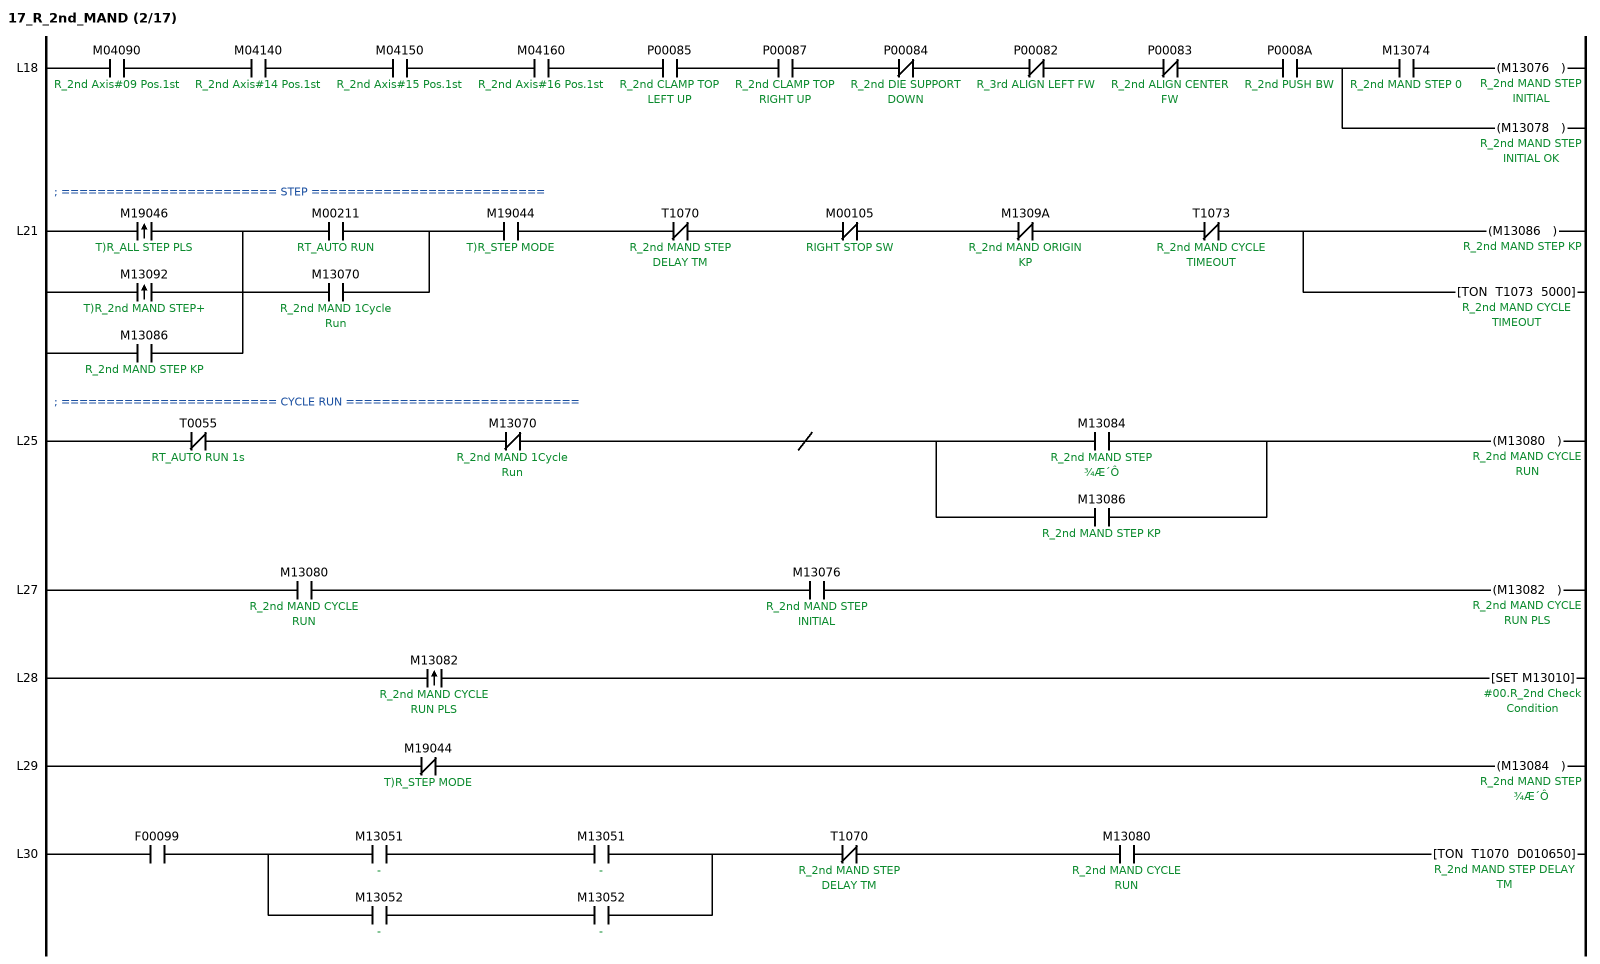
[picture p144: 17_R_2nd_MAND rungs L18-L30]
; L18
LOAD      M04090	// R_2nd Axis#09 Pos.1st
AND       M04140	// R_2nd Axis#14 Pos.1st
AND       M04150	// R_2nd Axis#15 Pos.1st
AND       M04160	// R_2nd Axis#16 Pos.1st
AND       P00085	// R_2nd CLAMP TOP LEFT UP
AND       P00087	// R_2nd CLAMP TOP RIGHT UP
AND NOT   P00084	// R_2nd DIE SUPPORT DOWN
AND NOT   P00082	// R_3rd ALIGN LEFT FW
AND NOT   P00083	// R_2nd ALIGN CENTER FW
AND       P0008A	// R_2nd PUSH BW
MPUSH
AND       M13074	// R_2nd MAND STEP 0
OUT       M13076	// R_2nd MAND STEP INITIAL
MPOP
OUT       M13078	// R_2nd MAND STEP INITIAL OK
// ======================== STEP ==========================
; L21
LOADP     M19046	// T)R_ALL STEP PLS
ORP       M13092	// T)R_2nd MAND STEP+
OR        M13086	// R_2nd MAND STEP KP
LOAD      M00211	// RT_AUTO RUN
OR        M13070	// R_2nd MAND 1Cycle Run
AND LOAD
AND       M19044	// T)R_STEP MODE
AND NOT   T1070	// R_2nd MAND STEP DELAY TM
AND NOT   M00105	// RIGHT STOP SW
AND NOT   M1309A	// R_2nd MAND ORIGIN KP
AND NOT   T1073	// R_2nd MAND CYCLE TIMEOUT
OUT       M13086	// R_2nd MAND STEP KP
TON       T1073 5000	// R_2nd MAND CYCLE TIMEOUT
// ======================== CYCLE RUN ==========================
; L25
LOAD NOT  T0055	// RT_AUTO RUN 1s
AND NOT   M13070	// R_2nd MAND 1Cycle Run
NOT
LOAD      M13084	// R_2nd MAND STEP ¾Æ´Ô
OR        M13086	// R_2nd MAND STEP KP
AND LOAD
OUT       M13080	// R_2nd MAND CYCLE RUN
; L27
LOAD      M13080	// R_2nd MAND CYCLE RUN
AND       M13076	// R_2nd MAND STEP INITIAL
OUT       M13082	// R_2nd MAND CYCLE RUN PLS
; L28
LOADP     M13082	// R_2nd MAND CYCLE RUN PLS
SET       M13010	// #00.R_2nd Check Condition
; L29
LOAD NOT  M19044	// T)R_STEP MODE
OUT       M13084	// R_2nd MAND STEP ¾Æ´Ô
; L30
LOAD      F00099
LOAD      M13051	// -
AND       M13051	// -
LOAD      M13052	// -
AND       M13052	// -
OR LOAD
AND LOAD
AND NOT   T1070	// R_2nd MAND STEP DELAY TM
AND       M13080	// R_2nd MAND CYCLE RUN
TON       T1070 D010650	// R_2nd MAND STEP DELAY TM

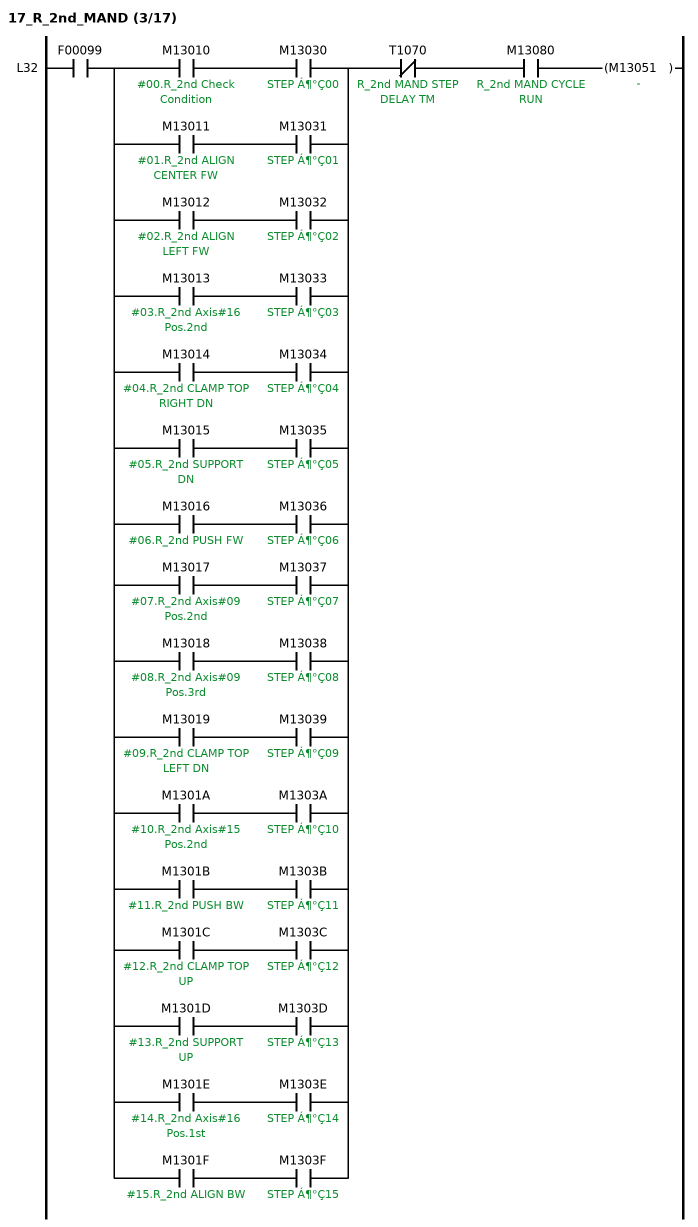
; L32
LOAD      F00099
LOAD      M13010	// #00.R_2nd Check Condition
AND       M13030	// STEP Á¶°Ç00
LOAD      M13011	// #01.R_2nd ALIGN CENTER FW
AND       M13031	// STEP Á¶°Ç01
OR LOAD
LOAD      M13012	// #02.R_2nd ALIGN LEFT FW
AND       M13032	// STEP Á¶°Ç02
OR LOAD
LOAD      M13013	// #03.R_2nd Axis#16 Pos.2nd
AND       M13033	// STEP Á¶°Ç03
OR LOAD
LOAD      M13014	// #04.R_2nd CLAMP TOP RIGHT DN
AND       M13034	// STEP Á¶°Ç04
OR LOAD
LOAD      M13015	// #05.R_2nd SUPPORT DN
AND       M13035	// STEP Á¶°Ç05
OR LOAD
LOAD      M13016	// #06.R_2nd PUSH FW
AND       M13036	// STEP Á¶°Ç06
OR LOAD
LOAD      M13017	// #07.R_2nd Axis#09 Pos.2nd
AND       M13037	// STEP Á¶°Ç07
OR LOAD
LOAD      M13018	// #08.R_2nd Axis#09 Pos.3rd
AND       M13038	// STEP Á¶°Ç08
OR LOAD
LOAD      M13019	// #09.R_2nd CLAMP TOP LEFT DN
AND       M13039	// STEP Á¶°Ç09
OR LOAD
LOAD      M1301A	// #10.R_2nd Axis#15 Pos.2nd
AND       M1303A	// STEP Á¶°Ç10
OR LOAD
LOAD      M1301B	// #11.R_2nd PUSH BW
AND       M1303B	// STEP Á¶°Ç11
OR LOAD
LOAD      M1301C	// #12.R_2nd CLAMP TOP UP
AND       M1303C	// STEP Á¶°Ç12
OR LOAD
LOAD      M1301D	// #13.R_2nd SUPPORT UP
AND       M1303D	// STEP Á¶°Ç13
OR LOAD
LOAD      M1301E	// #14.R_2nd Axis#16 Pos.1st
AND       M1303E	// STEP Á¶°Ç14
OR LOAD
LOAD      M1301F	// #15.R_2nd ALIGN BW
AND       M1303F	// STEP Á¶°Ç15
OR LOAD
AND LOAD
AND NOT   T1070	// R_2nd MAND STEP DELAY TM
AND       M13080	// R_2nd MAND CYCLE RUN
OUT       M13051	// -

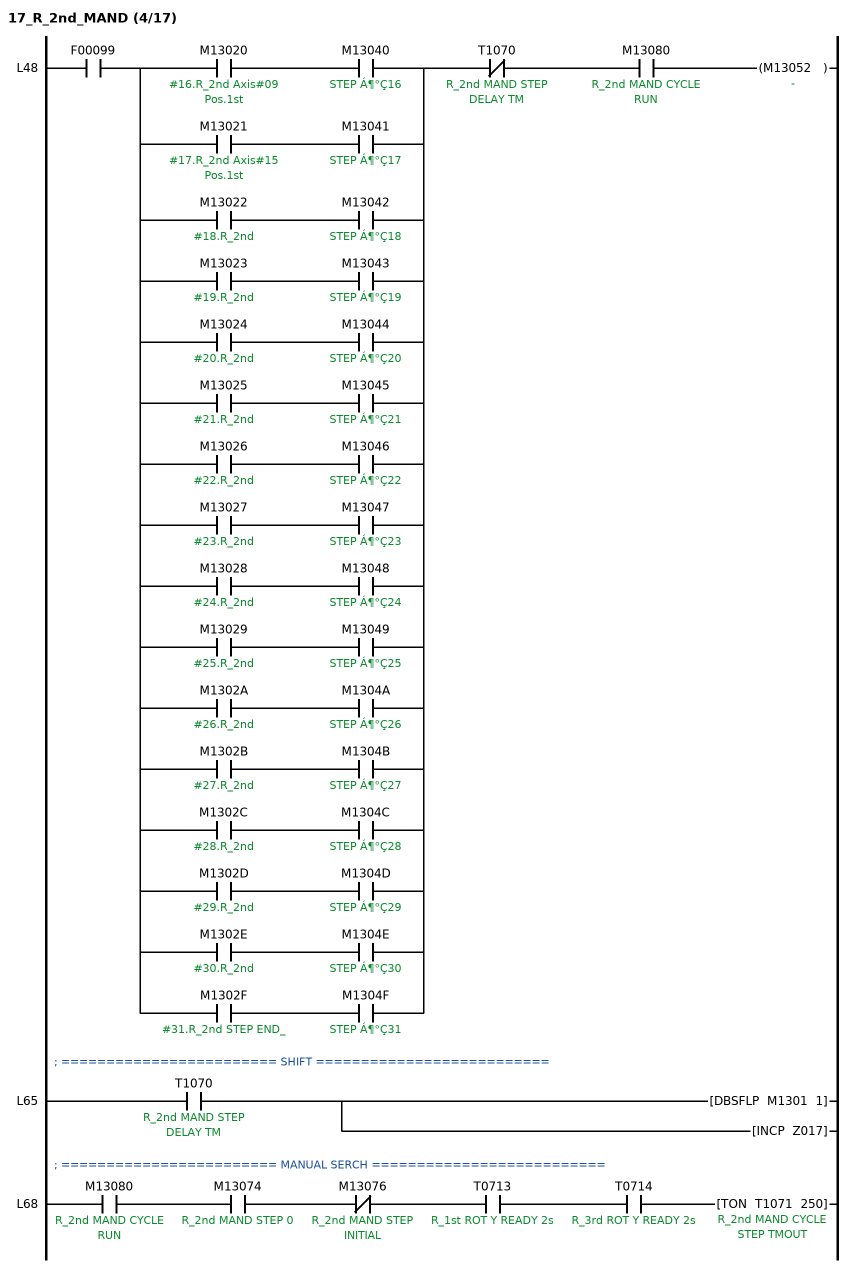
; L48
LOAD      F00099
LOAD      M13020	// #16.R_2nd Axis#09 Pos.1st
AND       M13040	// STEP Á¶°Ç16
LOAD      M13021	// #17.R_2nd Axis#15 Pos.1st
AND       M13041	// STEP Á¶°Ç17
OR LOAD
LOAD      M13022	// #18.R_2nd
AND       M13042	// STEP Á¶°Ç18
OR LOAD
LOAD      M13023	// #19.R_2nd
AND       M13043	// STEP Á¶°Ç19
OR LOAD
LOAD      M13024	// #20.R_2nd
AND       M13044	// STEP Á¶°Ç20
OR LOAD
LOAD      M13025	// #21.R_2nd
AND       M13045	// STEP Á¶°Ç21
OR LOAD
LOAD      M13026	// #22.R_2nd
AND       M13046	// STEP Á¶°Ç22
OR LOAD
LOAD      M13027	// #23.R_2nd
AND       M13047	// STEP Á¶°Ç23
OR LOAD
LOAD      M13028	// #24.R_2nd
AND       M13048	// STEP Á¶°Ç24
OR LOAD
LOAD      M13029	// #25.R_2nd
AND       M13049	// STEP Á¶°Ç25
OR LOAD
LOAD      M1302A	// #26.R_2nd
AND       M1304A	// STEP Á¶°Ç26
OR LOAD
LOAD      M1302B	// #27.R_2nd
AND       M1304B	// STEP Á¶°Ç27
OR LOAD
LOAD      M1302C	// #28.R_2nd
AND       M1304C	// STEP Á¶°Ç28
OR LOAD
LOAD      M1302D	// #29.R_2nd
AND       M1304D	// STEP Á¶°Ç29
OR LOAD
LOAD      M1302E	// #30.R_2nd
AND       M1304E	// STEP Á¶°Ç30
OR LOAD
LOAD      M1302F	// #31.R_2nd STEP END_
AND       M1304F	// STEP Á¶°Ç31
OR LOAD
AND LOAD
AND NOT   T1070	// R_2nd MAND STEP DELAY TM
AND       M13080	// R_2nd MAND CYCLE RUN
OUT       M13052	// -
// ======================== SHIFT ==========================
; L65
LOAD      T1070	// R_2nd MAND STEP DELAY TM
DBSFLP    M1301 1
INCP      Z017
// ======================== MANUAL SERCH ==========================
; L68
LOAD      M13080	// R_2nd MAND CYCLE RUN
AND       M13074	// R_2nd MAND STEP 0
AND NOT   M13076	// R_2nd MAND STEP INITIAL
AND       T0713	// R_1st ROT Y READY 2s
AND       T0714	// R_3rd ROT Y READY 2s
TON       T1071 250	// R_2nd MAND CYCLE STEP TMOUT

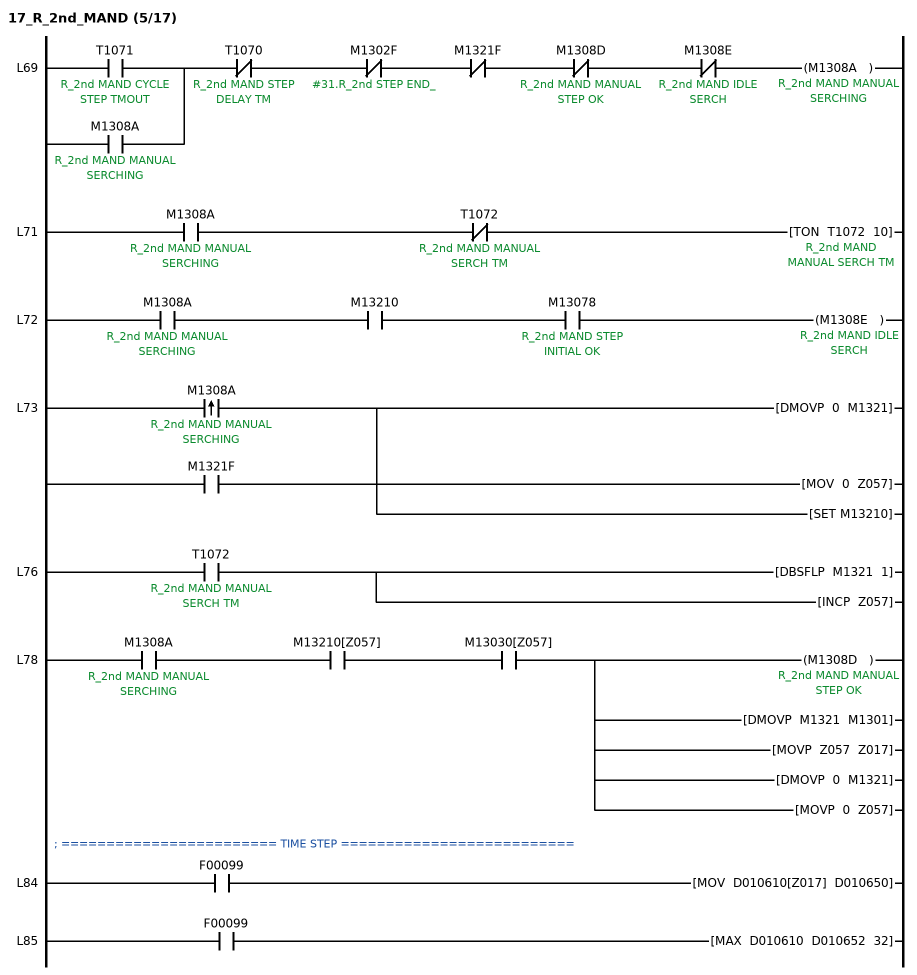
; L69
LOAD      T1071	// R_2nd MAND CYCLE STEP TMOUT
OR        M1308A	// R_2nd MAND MANUAL SERCHING
AND NOT   T1070	// R_2nd MAND STEP DELAY TM
AND NOT   M1302F	// #31.R_2nd STEP END_
AND NOT   M1321F
AND NOT   M1308D	// R_2nd MAND MANUAL STEP OK
AND NOT   M1308E	// R_2nd MAND IDLE SERCH
OUT       M1308A	// R_2nd MAND MANUAL SERCHING
; L71
LOAD      M1308A	// R_2nd MAND MANUAL SERCHING
AND NOT   T1072	// R_2nd MAND MANUAL SERCH TM
TON       T1072 10	// R_2nd MAND MANUAL SERCH TM
; L72
LOAD      M1308A	// R_2nd MAND MANUAL SERCHING
AND       M13210
AND       M13078	// R_2nd MAND STEP INITIAL OK
OUT       M1308E	// R_2nd MAND IDLE SERCH
; L73
LOADP     M1308A	// R_2nd MAND MANUAL SERCHING
OR        M1321F
DMOVP     0 M1321
MOV       0 Z057
SET       M13210
; L76
LOAD      T1072	// R_2nd MAND MANUAL SERCH TM
DBSFLP    M1321 1
INCP      Z057
; L78
LOAD      M1308A	// R_2nd MAND MANUAL SERCHING
AND       M13210[Z057]
AND       M13030[Z057]
OUT       M1308D	// R_2nd MAND MANUAL STEP OK
DMOVP     M1321 M1301
MOVP      Z057 Z017
DMOVP     0 M1321
MOVP      0 Z057
// ======================== TIME STEP ==========================
; L84
LOAD      F00099
MOV       D010610[Z017] D010650
; L85
LOAD      F00099
MAX       D010610 D010652 32

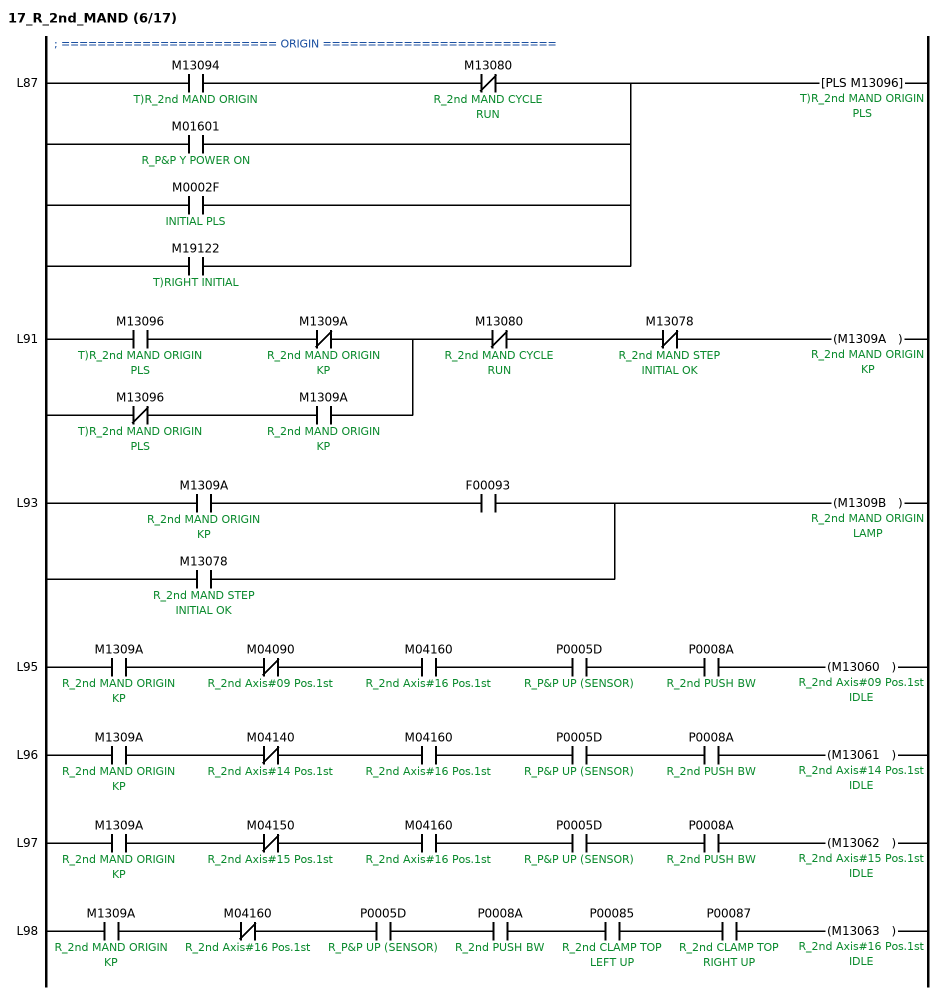
// ======================== ORIGIN ==========================
; L87
LOAD      M13094	// T)R_2nd MAND ORIGIN
AND NOT   M13080	// R_2nd MAND CYCLE RUN
OR        M01601	// R_P&P Y POWER ON
OR        M0002F	// INITIAL PLS
OR        M19122	// T)RIGHT INITIAL
OUTP      M13096	// T)R_2nd MAND ORIGIN PLS
; L91
LOAD      M13096	// T)R_2nd MAND ORIGIN PLS
AND NOT   M1309A	// R_2nd MAND ORIGIN KP
LOAD NOT  M13096	// T)R_2nd MAND ORIGIN PLS
AND       M1309A	// R_2nd MAND ORIGIN KP
OR LOAD
AND NOT   M13080	// R_2nd MAND CYCLE RUN
AND NOT   M13078	// R_2nd MAND STEP INITIAL OK
OUT       M1309A	// R_2nd MAND ORIGIN KP
; L93
LOAD      M1309A	// R_2nd MAND ORIGIN KP
AND       F00093
OR        M13078	// R_2nd MAND STEP INITIAL OK
OUT       M1309B	// R_2nd MAND ORIGIN LAMP
; L95
LOAD      M1309A	// R_2nd MAND ORIGIN KP
AND NOT   M04090	// R_2nd Axis#09 Pos.1st
AND       M04160	// R_2nd Axis#16 Pos.1st
AND       P0005D	// R_P&P UP (SENSOR)
AND       P0008A	// R_2nd PUSH BW
OUT       M13060	// R_2nd Axis#09 Pos.1st IDLE
; L96
LOAD      M1309A	// R_2nd MAND ORIGIN KP
AND NOT   M04140	// R_2nd Axis#14 Pos.1st
AND       M04160	// R_2nd Axis#16 Pos.1st
AND       P0005D	// R_P&P UP (SENSOR)
AND       P0008A	// R_2nd PUSH BW
OUT       M13061	// R_2nd Axis#14 Pos.1st IDLE
; L97
LOAD      M1309A	// R_2nd MAND ORIGIN KP
AND NOT   M04150	// R_2nd Axis#15 Pos.1st
AND       M04160	// R_2nd Axis#16 Pos.1st
AND       P0005D	// R_P&P UP (SENSOR)
AND       P0008A	// R_2nd PUSH BW
OUT       M13062	// R_2nd Axis#15 Pos.1st IDLE
; L98
LOAD      M1309A	// R_2nd MAND ORIGIN KP
AND NOT   M04160	// R_2nd Axis#16 Pos.1st
AND       P0005D	// R_P&P UP (SENSOR)
AND       P0008A	// R_2nd PUSH BW
AND       P00085	// R_2nd CLAMP TOP LEFT UP
AND       P00087	// R_2nd CLAMP TOP RIGHT UP
OUT       M13063	// R_2nd Axis#16 Pos.1st IDLE

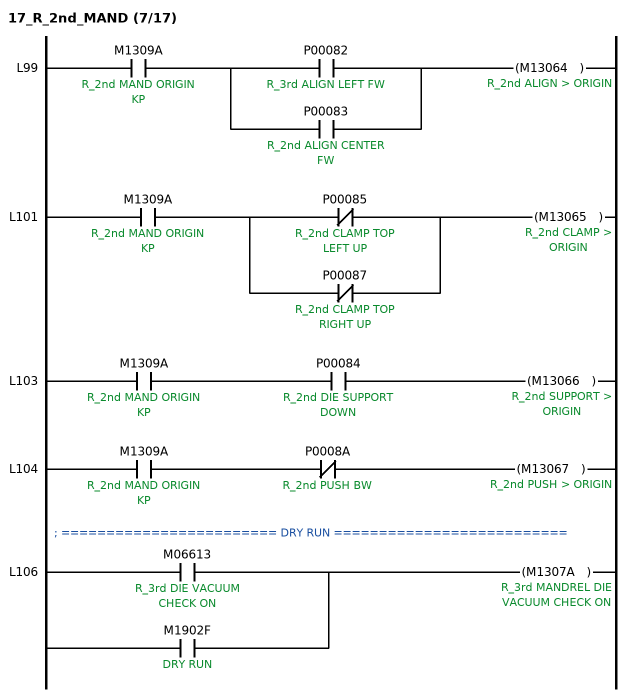
; L99
LOAD      M1309A	// R_2nd MAND ORIGIN KP
LOAD      P00082	// R_3rd ALIGN LEFT FW
OR        P00083	// R_2nd ALIGN CENTER FW
AND LOAD
OUT       M13064	// R_2nd ALIGN > ORIGIN
; L101
LOAD      M1309A	// R_2nd MAND ORIGIN KP
LOAD NOT  P00085	// R_2nd CLAMP TOP LEFT UP
OR NOT    P00087	// R_2nd CLAMP TOP RIGHT UP
AND LOAD
OUT       M13065	// R_2nd CLAMP > ORIGIN
; L103
LOAD      M1309A	// R_2nd MAND ORIGIN KP
AND       P00084	// R_2nd DIE SUPPORT DOWN
OUT       M13066	// R_2nd SUPPORT > ORIGIN
; L104
LOAD      M1309A	// R_2nd MAND ORIGIN KP
AND NOT   P0008A	// R_2nd PUSH BW
OUT       M13067	// R_2nd PUSH > ORIGIN
// ======================== DRY RUN ==========================
; L106
LOAD      M06613	// R_3rd DIE VACUUM CHECK ON
OR        M1902F	// DRY RUN
OUT       M1307A	// R_3rd MANDREL DIE VACUUM CHECK ON

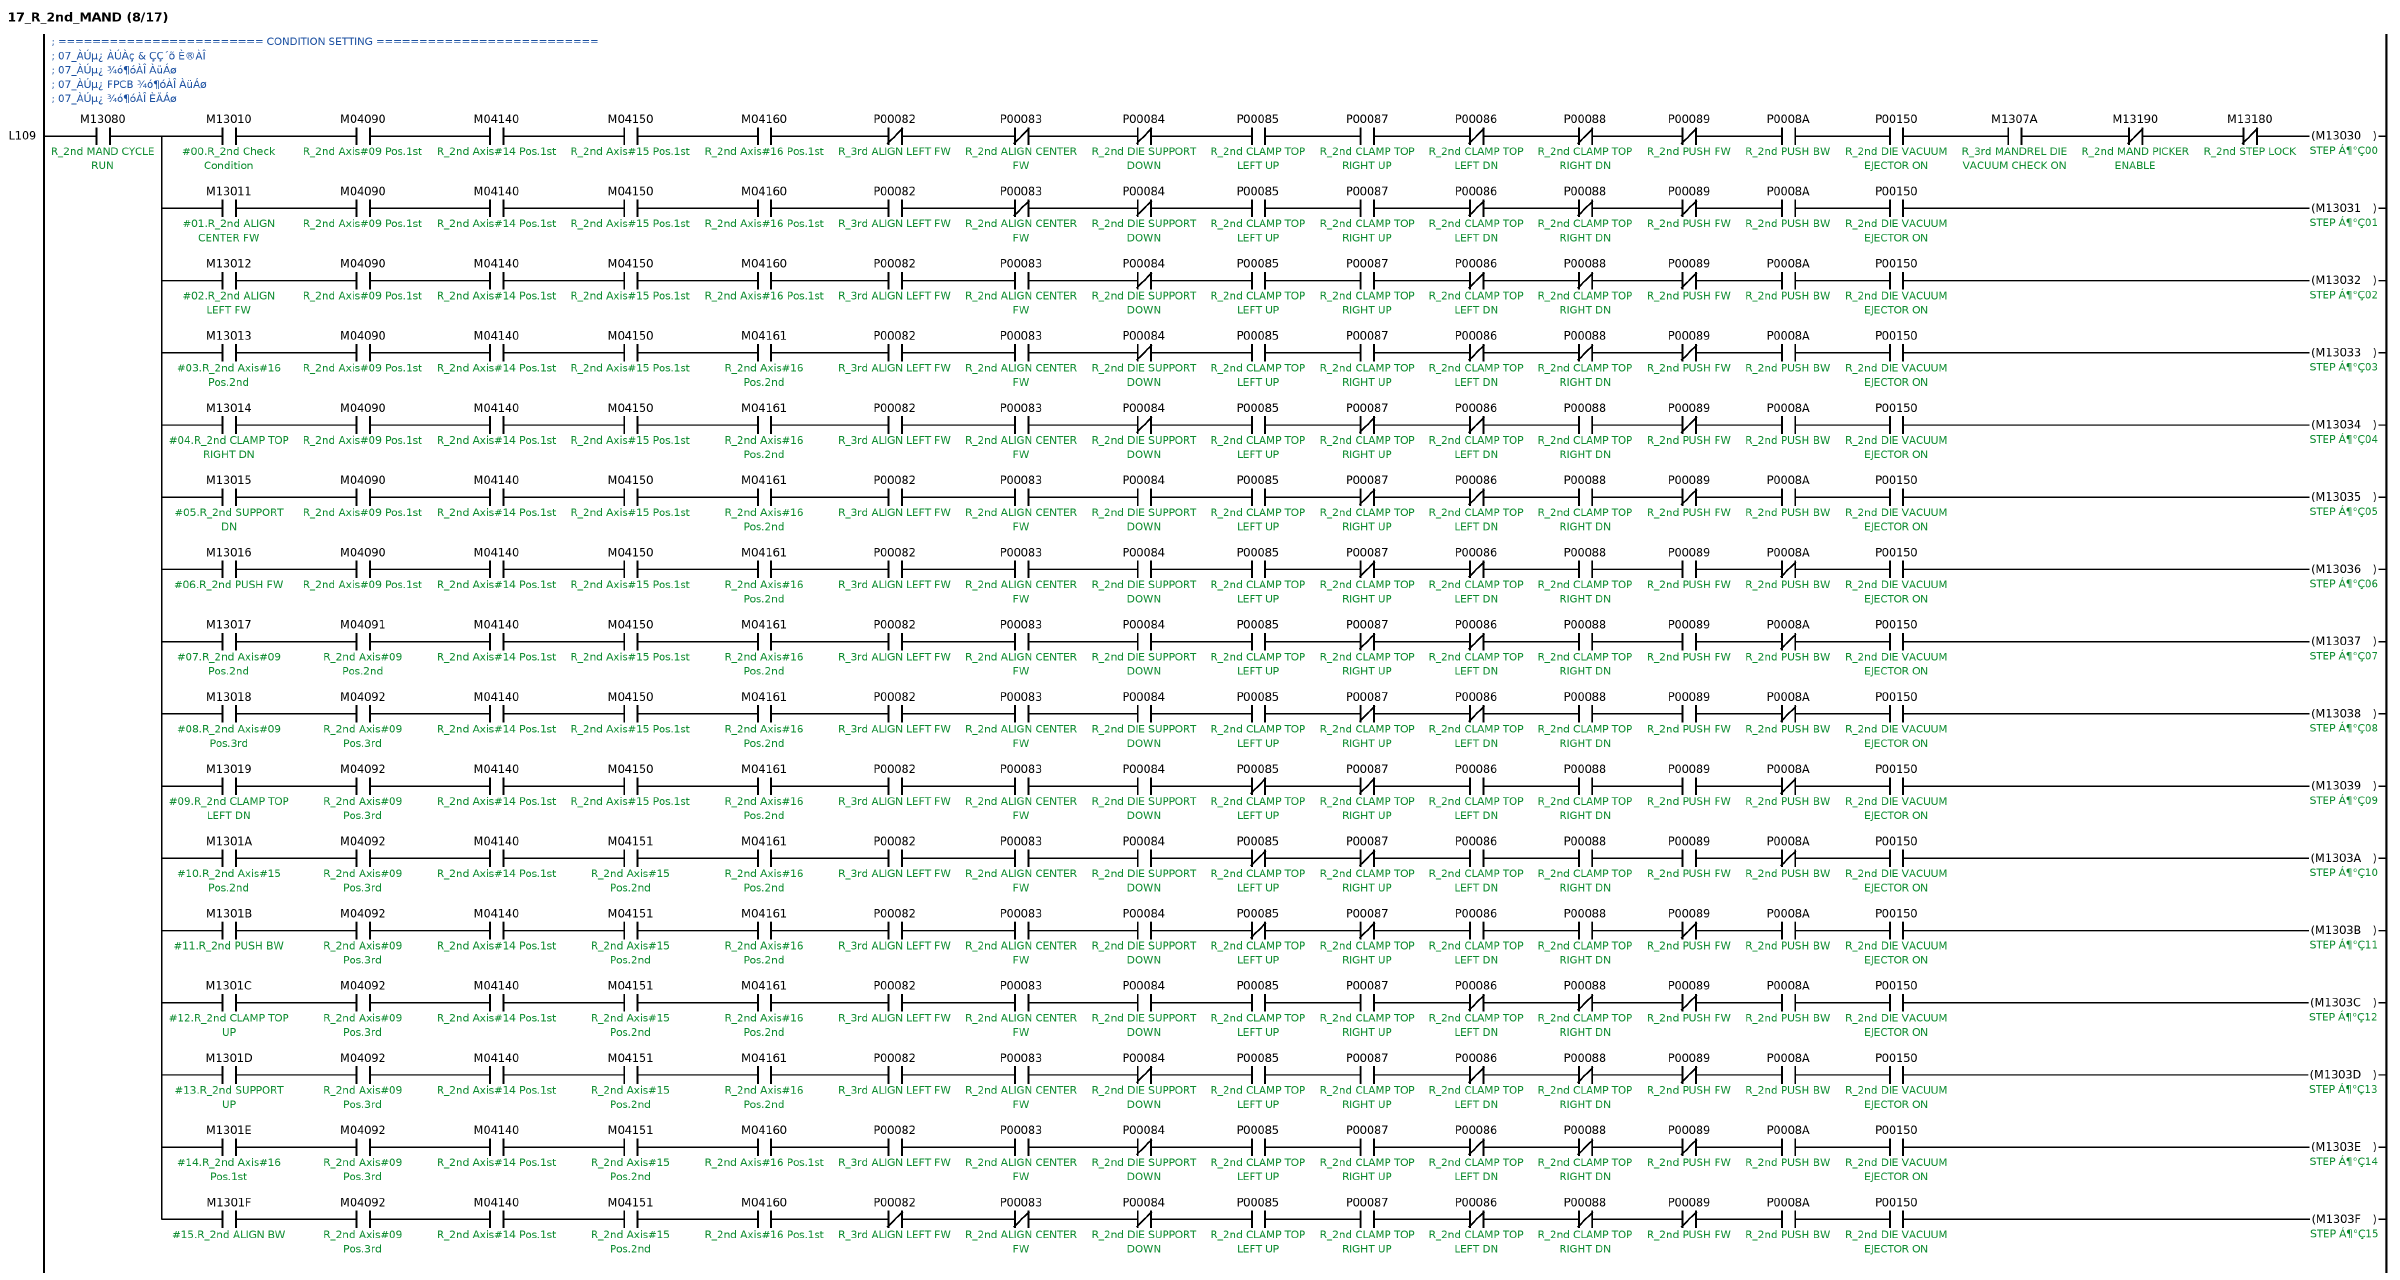
// ======================== CONDITION SETTING ==========================
; L109
LOAD      M13080	// R_2nd MAND CYCLE RUN
MPUSH
AND       M13010	// #00.R_2nd Check Condition
AND       M04090	// R_2nd Axis#09 Pos.1st
AND       M04140	// R_2nd Axis#14 Pos.1st
AND       M04150	// R_2nd Axis#15 Pos.1st
AND       M04160	// R_2nd Axis#16 Pos.1st
AND NOT   P00082	// R_3rd ALIGN LEFT FW
AND NOT   P00083	// R_2nd ALIGN CENTER FW
AND NOT   P00084	// R_2nd DIE SUPPORT DOWN
AND       P00085	// R_2nd CLAMP TOP LEFT UP
AND       P00087	// R_2nd CLAMP TOP RIGHT UP
AND NOT   P00086	// R_2nd CLAMP TOP LEFT DN
AND NOT   P00088	// R_2nd CLAMP TOP RIGHT DN
AND NOT   P00089	// R_2nd PUSH FW
AND       P0008A	// R_2nd PUSH BW
AND       P00150	// R_2nd DIE VACUUM EJECTOR ON
AND       M1307A	// R_3rd MANDREL DIE VACUUM CHECK ON
AND NOT   M13190	// R_2nd MAND PICKER ENABLE
AND NOT   M13180	// R_2nd STEP LOCK
OUT       M13030	// STEP Á¶°Ç00
MLOAD
AND       M13011	// #01.R_2nd ALIGN CENTER FW
AND       M04090	// R_2nd Axis#09 Pos.1st
AND       M04140	// R_2nd Axis#14 Pos.1st
AND       M04150	// R_2nd Axis#15 Pos.1st
AND       M04160	// R_2nd Axis#16 Pos.1st
AND       P00082	// R_3rd ALIGN LEFT FW
AND NOT   P00083	// R_2nd ALIGN CENTER FW
AND NOT   P00084	// R_2nd DIE SUPPORT DOWN
AND       P00085	// R_2nd CLAMP TOP LEFT UP
AND       P00087	// R_2nd CLAMP TOP RIGHT UP
AND NOT   P00086	// R_2nd CLAMP TOP LEFT DN
AND NOT   P00088	// R_2nd CLAMP TOP RIGHT DN
AND NOT   P00089	// R_2nd PUSH FW
AND       P0008A	// R_2nd PUSH BW
AND       P00150	// R_2nd DIE VACUUM EJECTOR ON
OUT       M13031	// STEP Á¶°Ç01
MLOAD
AND       M13012	// #02.R_2nd ALIGN LEFT FW
AND       M04090	// R_2nd Axis#09 Pos.1st
AND       M04140	// R_2nd Axis#14 Pos.1st
AND       M04150	// R_2nd Axis#15 Pos.1st
AND       M04160	// R_2nd Axis#16 Pos.1st
AND       P00082	// R_3rd ALIGN LEFT FW
AND       P00083	// R_2nd ALIGN CENTER FW
AND NOT   P00084	// R_2nd DIE SUPPORT DOWN
AND       P00085	// R_2nd CLAMP TOP LEFT UP
AND       P00087	// R_2nd CLAMP TOP RIGHT UP
AND NOT   P00086	// R_2nd CLAMP TOP LEFT DN
AND NOT   P00088	// R_2nd CLAMP TOP RIGHT DN
AND NOT   P00089	// R_2nd PUSH FW
AND       P0008A	// R_2nd PUSH BW
AND       P00150	// R_2nd DIE VACUUM EJECTOR ON
OUT       M13032	// STEP Á¶°Ç02
MLOAD
AND       M13013	// #03.R_2nd Axis#16 Pos.2nd
AND       M04090	// R_2nd Axis#09 Pos.1st
AND       M04140	// R_2nd Axis#14 Pos.1st
AND       M04150	// R_2nd Axis#15 Pos.1st
AND       M04161	// R_2nd Axis#16 Pos.2nd
AND       P00082	// R_3rd ALIGN LEFT FW
AND       P00083	// R_2nd ALIGN CENTER FW
AND NOT   P00084	// R_2nd DIE SUPPORT DOWN
AND       P00085	// R_2nd CLAMP TOP LEFT UP
AND       P00087	// R_2nd CLAMP TOP RIGHT UP
AND NOT   P00086	// R_2nd CLAMP TOP LEFT DN
AND NOT   P00088	// R_2nd CLAMP TOP RIGHT DN
AND NOT   P00089	// R_2nd PUSH FW
AND       P0008A	// R_2nd PUSH BW
AND       P00150	// R_2nd DIE VACUUM EJECTOR ON
OUT       M13033	// STEP Á¶°Ç03
MLOAD
AND       M13014	// #04.R_2nd CLAMP TOP RIGHT DN
AND       M04090	// R_2nd Axis#09 Pos.1st
AND       M04140	// R_2nd Axis#14 Pos.1st
AND       M04150	// R_2nd Axis#15 Pos.1st
AND       M04161	// R_2nd Axis#16 Pos.2nd
AND       P00082	// R_3rd ALIGN LEFT FW
AND       P00083	// R_2nd ALIGN CENTER FW
AND NOT   P00084	// R_2nd DIE SUPPORT DOWN
AND       P00085	// R_2nd CLAMP TOP LEFT UP
AND NOT   P00087	// R_2nd CLAMP TOP RIGHT UP
AND NOT   P00086	// R_2nd CLAMP TOP LEFT DN
AND       P00088	// R_2nd CLAMP TOP RIGHT DN
AND NOT   P00089	// R_2nd PUSH FW
AND       P0008A	// R_2nd PUSH BW
AND       P00150	// R_2nd DIE VACUUM EJECTOR ON
OUT       M13034	// STEP Á¶°Ç04
MLOAD
AND       M13015	// #05.R_2nd SUPPORT DN
AND       M04090	// R_2nd Axis#09 Pos.1st
AND       M04140	// R_2nd Axis#14 Pos.1st
AND       M04150	// R_2nd Axis#15 Pos.1st
AND       M04161	// R_2nd Axis#16 Pos.2nd
AND       P00082	// R_3rd ALIGN LEFT FW
AND       P00083	// R_2nd ALIGN CENTER FW
AND       P00084	// R_2nd DIE SUPPORT DOWN
AND       P00085	// R_2nd CLAMP TOP LEFT UP
AND NOT   P00087	// R_2nd CLAMP TOP RIGHT UP
AND NOT   P00086	// R_2nd CLAMP TOP LEFT DN
AND       P00088	// R_2nd CLAMP TOP RIGHT DN
AND NOT   P00089	// R_2nd PUSH FW
AND       P0008A	// R_2nd PUSH BW
AND       P00150	// R_2nd DIE VACUUM EJECTOR ON
OUT       M13035	// STEP Á¶°Ç05
MLOAD
AND       M13016	// #06.R_2nd PUSH FW
AND       M04090	// R_2nd Axis#09 Pos.1st
AND       M04140	// R_2nd Axis#14 Pos.1st
AND       M04150	// R_2nd Axis#15 Pos.1st
AND       M04161	// R_2nd Axis#16 Pos.2nd
AND       P00082	// R_3rd ALIGN LEFT FW
AND       P00083	// R_2nd ALIGN CENTER FW
AND       P00084	// R_2nd DIE SUPPORT DOWN
AND       P00085	// R_2nd CLAMP TOP LEFT UP
AND NOT   P00087	// R_2nd CLAMP TOP RIGHT UP
AND NOT   P00086	// R_2nd CLAMP TOP LEFT DN
AND       P00088	// R_2nd CLAMP TOP RIGHT DN
AND       P00089	// R_2nd PUSH FW
AND NOT   P0008A	// R_2nd PUSH BW
AND       P00150	// R_2nd DIE VACUUM EJECTOR ON
OUT       M13036	// STEP Á¶°Ç06
MLOAD
AND       M13017	// #07.R_2nd Axis#09 Pos.2nd
AND       M04091	// R_2nd Axis#09 Pos.2nd
AND       M04140	// R_2nd Axis#14 Pos.1st
AND       M04150	// R_2nd Axis#15 Pos.1st
AND       M04161	// R_2nd Axis#16 Pos.2nd
AND       P00082	// R_3rd ALIGN LEFT FW
AND       P00083	// R_2nd ALIGN CENTER FW
AND       P00084	// R_2nd DIE SUPPORT DOWN
AND       P00085	// R_2nd CLAMP TOP LEFT UP
AND NOT   P00087	// R_2nd CLAMP TOP RIGHT UP
AND NOT   P00086	// R_2nd CLAMP TOP LEFT DN
AND       P00088	// R_2nd CLAMP TOP RIGHT DN
AND       P00089	// R_2nd PUSH FW
AND NOT   P0008A	// R_2nd PUSH BW
AND       P00150	// R_2nd DIE VACUUM EJECTOR ON
OUT       M13037	// STEP Á¶°Ç07
MLOAD
AND       M13018	// #08.R_2nd Axis#09 Pos.3rd
AND       M04092	// R_2nd Axis#09 Pos.3rd
AND       M04140	// R_2nd Axis#14 Pos.1st
AND       M04150	// R_2nd Axis#15 Pos.1st
AND       M04161	// R_2nd Axis#16 Pos.2nd
AND       P00082	// R_3rd ALIGN LEFT FW
AND       P00083	// R_2nd ALIGN CENTER FW
AND       P00084	// R_2nd DIE SUPPORT DOWN
AND       P00085	// R_2nd CLAMP TOP LEFT UP
AND NOT   P00087	// R_2nd CLAMP TOP RIGHT UP
AND NOT   P00086	// R_2nd CLAMP TOP LEFT DN
AND       P00088	// R_2nd CLAMP TOP RIGHT DN
AND       P00089	// R_2nd PUSH FW
AND NOT   P0008A	// R_2nd PUSH BW
AND       P00150	// R_2nd DIE VACUUM EJECTOR ON
OUT       M13038	// STEP Á¶°Ç08
MLOAD
AND       M13019	// #09.R_2nd CLAMP TOP LEFT DN
AND       M04092	// R_2nd Axis#09 Pos.3rd
AND       M04140	// R_2nd Axis#14 Pos.1st
AND       M04150	// R_2nd Axis#15 Pos.1st
AND       M04161	// R_2nd Axis#16 Pos.2nd
AND       P00082	// R_3rd ALIGN LEFT FW
AND       P00083	// R_2nd ALIGN CENTER FW
AND       P00084	// R_2nd DIE SUPPORT DOWN
AND NOT   P00085	// R_2nd CLAMP TOP LEFT UP
AND NOT   P00087	// R_2nd CLAMP TOP RIGHT UP
AND       P00086	// R_2nd CLAMP TOP LEFT DN
AND       P00088	// R_2nd CLAMP TOP RIGHT DN
AND       P00089	// R_2nd PUSH FW
AND NOT   P0008A	// R_2nd PUSH BW
AND       P00150	// R_2nd DIE VACUUM EJECTOR ON
OUT       M13039	// STEP Á¶°Ç09
MLOAD
AND       M1301A	// #10.R_2nd Axis#15 Pos.2nd
AND       M04092	// R_2nd Axis#09 Pos.3rd
AND       M04140	// R_2nd Axis#14 Pos.1st
AND       M04151	// R_2nd Axis#15 Pos.2nd
AND       M04161	// R_2nd Axis#16 Pos.2nd
AND       P00082	// R_3rd ALIGN LEFT FW
AND       P00083	// R_2nd ALIGN CENTER FW
AND       P00084	// R_2nd DIE SUPPORT DOWN
AND NOT   P00085	// R_2nd CLAMP TOP LEFT UP
AND NOT   P00087	// R_2nd CLAMP TOP RIGHT UP
AND       P00086	// R_2nd CLAMP TOP LEFT DN
AND       P00088	// R_2nd CLAMP TOP RIGHT DN
AND       P00089	// R_2nd PUSH FW
AND NOT   P0008A	// R_2nd PUSH BW
AND       P00150	// R_2nd DIE VACUUM EJECTOR ON
OUT       M1303A	// STEP Á¶°Ç10
MLOAD
AND       M1301B	// #11.R_2nd PUSH BW
AND       M04092	// R_2nd Axis#09 Pos.3rd
AND       M04140	// R_2nd Axis#14 Pos.1st
AND       M04151	// R_2nd Axis#15 Pos.2nd
AND       M04161	// R_2nd Axis#16 Pos.2nd
AND       P00082	// R_3rd ALIGN LEFT FW
AND       P00083	// R_2nd ALIGN CENTER FW
AND       P00084	// R_2nd DIE SUPPORT DOWN
AND NOT   P00085	// R_2nd CLAMP TOP LEFT UP
AND NOT   P00087	// R_2nd CLAMP TOP RIGHT UP
AND       P00086	// R_2nd CLAMP TOP LEFT DN
AND       P00088	// R_2nd CLAMP TOP RIGHT DN
AND NOT   P00089	// R_2nd PUSH FW
AND       P0008A	// R_2nd PUSH BW
AND       P00150	// R_2nd DIE VACUUM EJECTOR ON
OUT       M1303B	// STEP Á¶°Ç11
MLOAD
AND       M1301C	// #12.R_2nd CLAMP TOP UP
AND       M04092	// R_2nd Axis#09 Pos.3rd
AND       M04140	// R_2nd Axis#14 Pos.1st
AND       M04151	// R_2nd Axis#15 Pos.2nd
AND       M04161	// R_2nd Axis#16 Pos.2nd
AND       P00082	// R_3rd ALIGN LEFT FW
AND       P00083	// R_2nd ALIGN CENTER FW
AND       P00084	// R_2nd DIE SUPPORT DOWN
AND       P00085	// R_2nd CLAMP TOP LEFT UP
AND       P00087	// R_2nd CLAMP TOP RIGHT UP
AND NOT   P00086	// R_2nd CLAMP TOP LEFT DN
AND NOT   P00088	// R_2nd CLAMP TOP RIGHT DN
AND NOT   P00089	// R_2nd PUSH FW
AND       P0008A	// R_2nd PUSH BW
AND       P00150	// R_2nd DIE VACUUM EJECTOR ON
OUT       M1303C	// STEP Á¶°Ç12
MLOAD
AND       M1301D	// #13.R_2nd SUPPORT UP
AND       M04092	// R_2nd Axis#09 Pos.3rd
AND       M04140	// R_2nd Axis#14 Pos.1st
AND       M04151	// R_2nd Axis#15 Pos.2nd
AND       M04161	// R_2nd Axis#16 Pos.2nd
AND       P00082	// R_3rd ALIGN LEFT FW
AND       P00083	// R_2nd ALIGN CENTER FW
AND NOT   P00084	// R_2nd DIE SUPPORT DOWN
AND       P00085	// R_2nd CLAMP TOP LEFT UP
AND       P00087	// R_2nd CLAMP TOP RIGHT UP
AND NOT   P00086	// R_2nd CLAMP TOP LEFT DN
AND NOT   P00088	// R_2nd CLAMP TOP RIGHT DN
AND NOT   P00089	// R_2nd PUSH FW
AND       P0008A	// R_2nd PUSH BW
AND       P00150	// R_2nd DIE VACUUM EJECTOR ON
OUT       M1303D	// STEP Á¶°Ç13
MLOAD
AND       M1301E	// #14.R_2nd Axis#16 Pos.1st
AND       M04092	// R_2nd Axis#09 Pos.3rd
AND       M04140	// R_2nd Axis#14 Pos.1st
AND       M04151	// R_2nd Axis#15 Pos.2nd
AND       M04160	// R_2nd Axis#16 Pos.1st
AND       P00082	// R_3rd ALIGN LEFT FW
AND       P00083	// R_2nd ALIGN CENTER FW
AND NOT   P00084	// R_2nd DIE SUPPORT DOWN
AND       P00085	// R_2nd CLAMP TOP LEFT UP
AND       P00087	// R_2nd CLAMP TOP RIGHT UP
AND NOT   P00086	// R_2nd CLAMP TOP LEFT DN
AND NOT   P00088	// R_2nd CLAMP TOP RIGHT DN
AND NOT   P00089	// R_2nd PUSH FW
AND       P0008A	// R_2nd PUSH BW
AND       P00150	// R_2nd DIE VACUUM EJECTOR ON
OUT       M1303E	// STEP Á¶°Ç14
MPOP
AND       M1301F	// #15.R_2nd ALIGN BW
AND       M04092	// R_2nd Axis#09 Pos.3rd
AND       M04140	// R_2nd Axis#14 Pos.1st
AND       M04151	// R_2nd Axis#15 Pos.2nd
AND       M04160	// R_2nd Axis#16 Pos.1st
AND NOT   P00082	// R_3rd ALIGN LEFT FW
AND NOT   P00083	// R_2nd ALIGN CENTER FW
AND NOT   P00084	// R_2nd DIE SUPPORT DOWN
AND       P00085	// R_2nd CLAMP TOP LEFT UP
AND       P00087	// R_2nd CLAMP TOP RIGHT UP
AND NOT   P00086	// R_2nd CLAMP TOP LEFT DN
AND NOT   P00088	// R_2nd CLAMP TOP RIGHT DN
AND NOT   P00089	// R_2nd PUSH FW
AND       P0008A	// R_2nd PUSH BW
AND       P00150	// R_2nd DIE VACUUM EJECTOR ON
OUT       M1303F	// STEP Á¶°Ç15
// output comment: 07_ÀÚµ¿ ÀÚÀç & ÇÇ´õ È®ÀÎ
// output comment: 07_ÀÚµ¿ ¾ó¶óÀÎ ÀüÁø
// output comment: 07_ÀÚµ¿ FPCB ¾ó¶óÀÎ ÀüÁø
// output comment: 07_ÀÚµ¿ ¾ó¶óÀÎ ÈÄÁø

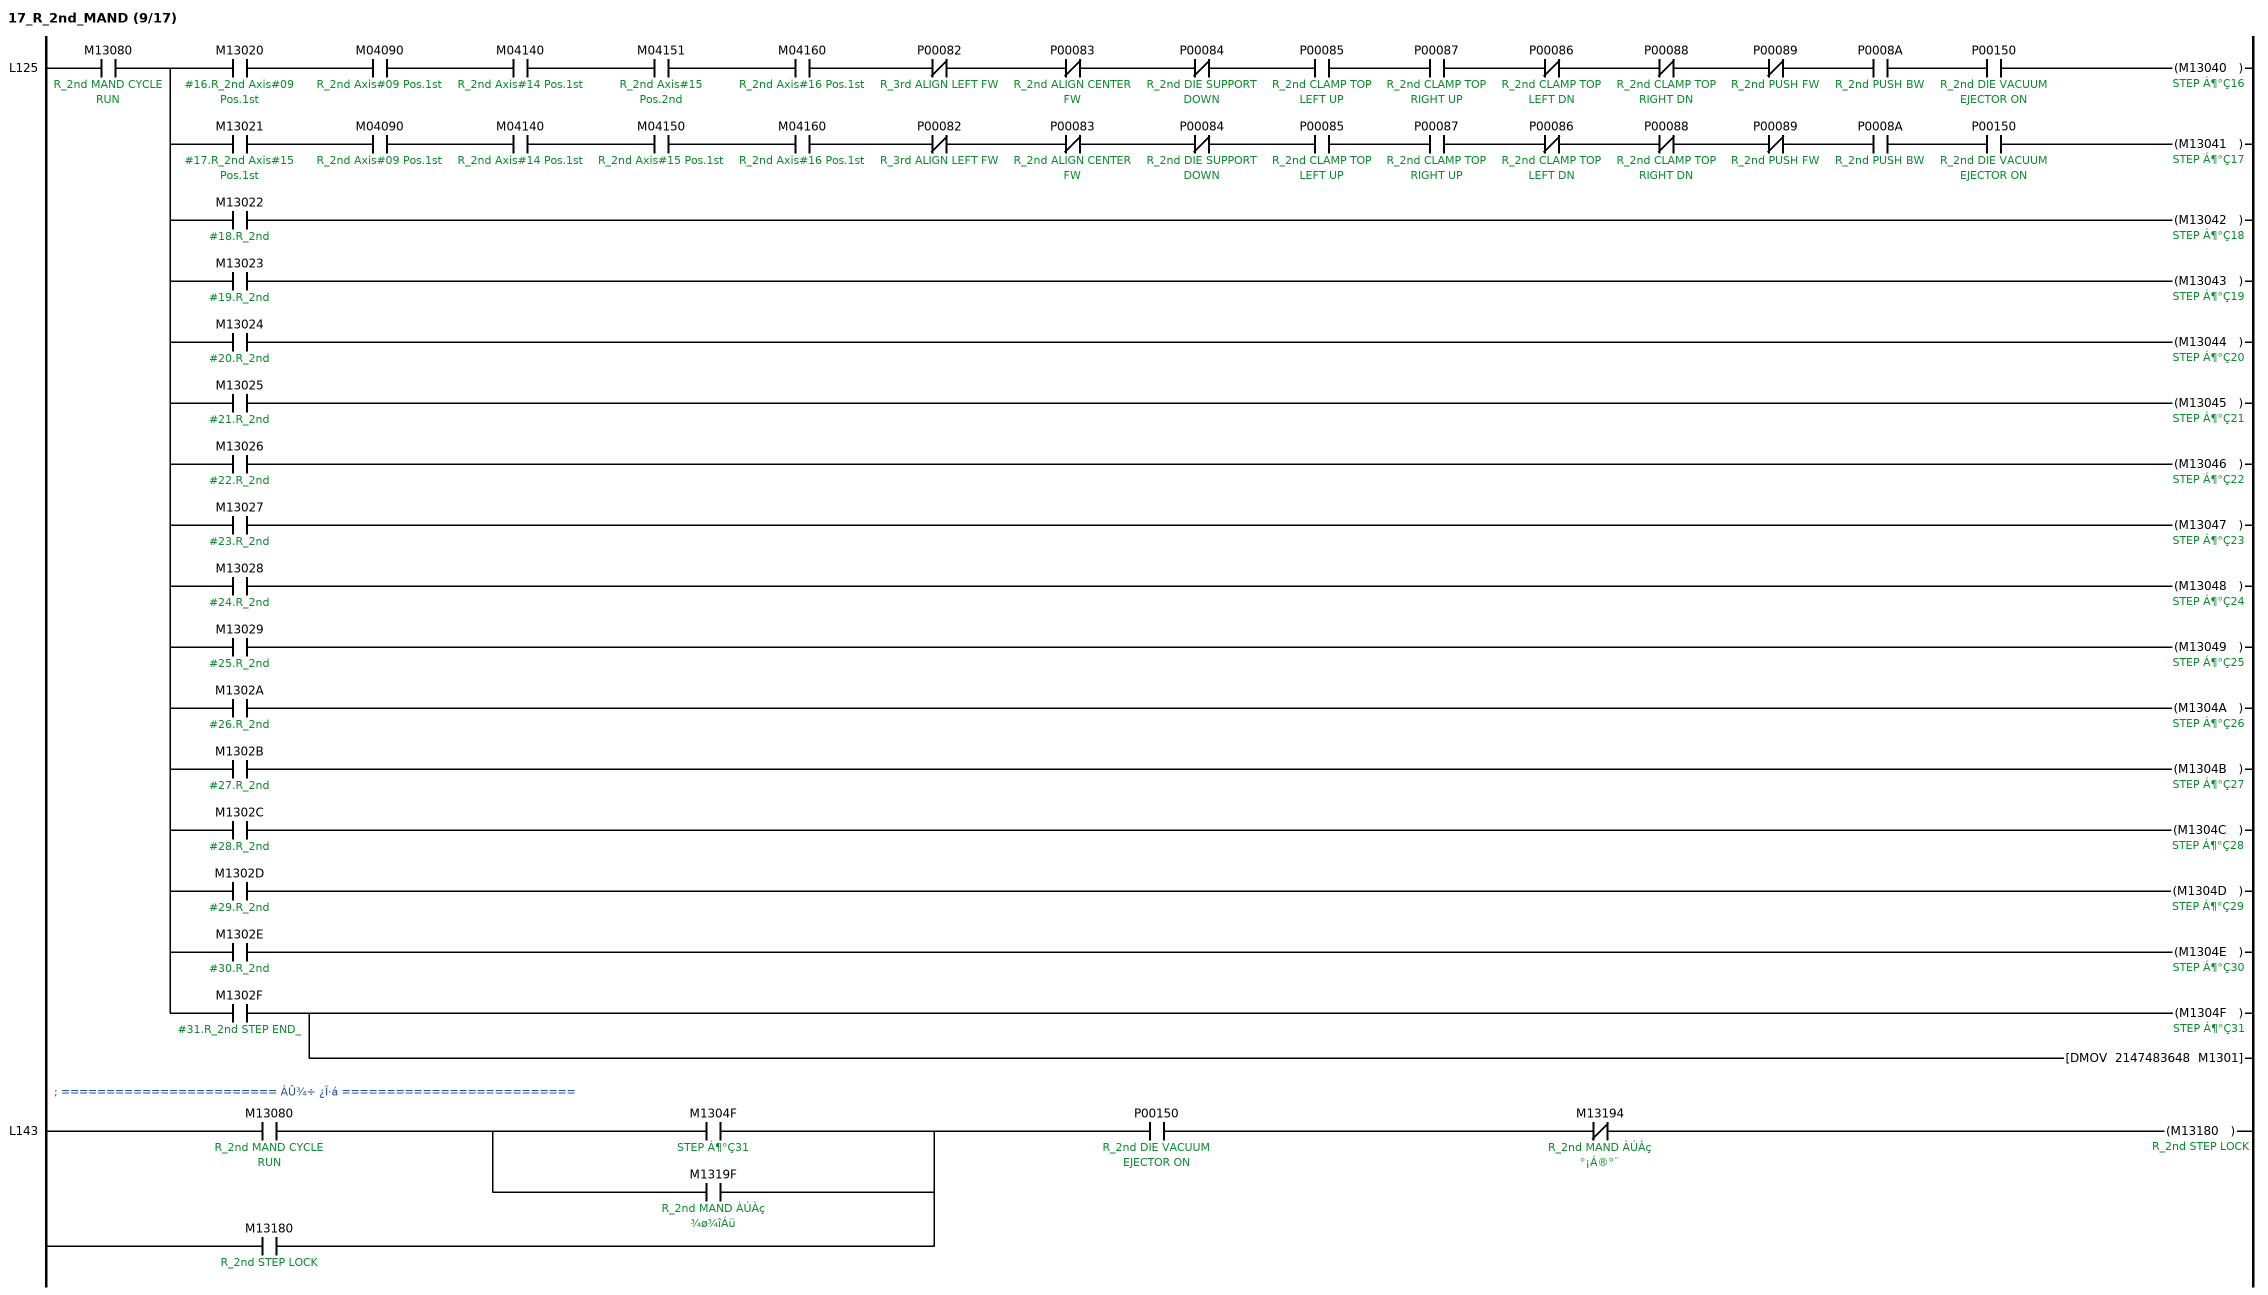
; L125
LOAD      M13080	// R_2nd MAND CYCLE RUN
MPUSH
AND       M13020	// #16.R_2nd Axis#09 Pos.1st
AND       M04090	// R_2nd Axis#09 Pos.1st
AND       M04140	// R_2nd Axis#14 Pos.1st
AND       M04151	// R_2nd Axis#15 Pos.2nd
AND       M04160	// R_2nd Axis#16 Pos.1st
AND NOT   P00082	// R_3rd ALIGN LEFT FW
AND NOT   P00083	// R_2nd ALIGN CENTER FW
AND NOT   P00084	// R_2nd DIE SUPPORT DOWN
AND       P00085	// R_2nd CLAMP TOP LEFT UP
AND       P00087	// R_2nd CLAMP TOP RIGHT UP
AND NOT   P00086	// R_2nd CLAMP TOP LEFT DN
AND NOT   P00088	// R_2nd CLAMP TOP RIGHT DN
AND NOT   P00089	// R_2nd PUSH FW
AND       P0008A	// R_2nd PUSH BW
AND       P00150	// R_2nd DIE VACUUM EJECTOR ON
OUT       M13040	// STEP Á¶°Ç16
MLOAD
AND       M13021	// #17.R_2nd Axis#15 Pos.1st
AND       M04090	// R_2nd Axis#09 Pos.1st
AND       M04140	// R_2nd Axis#14 Pos.1st
AND       M04150	// R_2nd Axis#15 Pos.1st
AND       M04160	// R_2nd Axis#16 Pos.1st
AND NOT   P00082	// R_3rd ALIGN LEFT FW
AND NOT   P00083	// R_2nd ALIGN CENTER FW
AND NOT   P00084	// R_2nd DIE SUPPORT DOWN
AND       P00085	// R_2nd CLAMP TOP LEFT UP
AND       P00087	// R_2nd CLAMP TOP RIGHT UP
AND NOT   P00086	// R_2nd CLAMP TOP LEFT DN
AND NOT   P00088	// R_2nd CLAMP TOP RIGHT DN
AND NOT   P00089	// R_2nd PUSH FW
AND       P0008A	// R_2nd PUSH BW
AND       P00150	// R_2nd DIE VACUUM EJECTOR ON
OUT       M13041	// STEP Á¶°Ç17
MLOAD
AND       M13022	// #18.R_2nd
OUT       M13042	// STEP Á¶°Ç18
MLOAD
AND       M13023	// #19.R_2nd
OUT       M13043	// STEP Á¶°Ç19
MLOAD
AND       M13024	// #20.R_2nd
OUT       M13044	// STEP Á¶°Ç20
MLOAD
AND       M13025	// #21.R_2nd
OUT       M13045	// STEP Á¶°Ç21
MLOAD
AND       M13026	// #22.R_2nd
OUT       M13046	// STEP Á¶°Ç22
MLOAD
AND       M13027	// #23.R_2nd
OUT       M13047	// STEP Á¶°Ç23
MLOAD
AND       M13028	// #24.R_2nd
OUT       M13048	// STEP Á¶°Ç24
MLOAD
AND       M13029	// #25.R_2nd
OUT       M13049	// STEP Á¶°Ç25
MLOAD
AND       M1302A	// #26.R_2nd
OUT       M1304A	// STEP Á¶°Ç26
MLOAD
AND       M1302B	// #27.R_2nd
OUT       M1304B	// STEP Á¶°Ç27
MLOAD
AND       M1302C	// #28.R_2nd
OUT       M1304C	// STEP Á¶°Ç28
MLOAD
AND       M1302D	// #29.R_2nd
OUT       M1304D	// STEP Á¶°Ç29
MLOAD
AND       M1302E	// #30.R_2nd
OUT       M1304E	// STEP Á¶°Ç30
MPOP
AND       M1302F	// #31.R_2nd STEP END_
OUT       M1304F	// STEP Á¶°Ç31
DMOV      2147483648 M1301
// ======================== ÀÛ¾÷ ¿Ï·á ==========================
; L143
LOAD      M13080	// R_2nd MAND CYCLE RUN
LOAD      M1304F	// STEP Á¶°Ç31
OR        M1319F	// R_2nd MAND ÀÚÀç ¾ø¾îÁü
AND LOAD
OR        M13180	// R_2nd STEP LOCK
AND       P00150	// R_2nd DIE VACUUM EJECTOR ON
AND NOT   M13194	// R_2nd MAND ÀÚÀç °¡Á®°¨
OUT       M13180	// R_2nd STEP LOCK

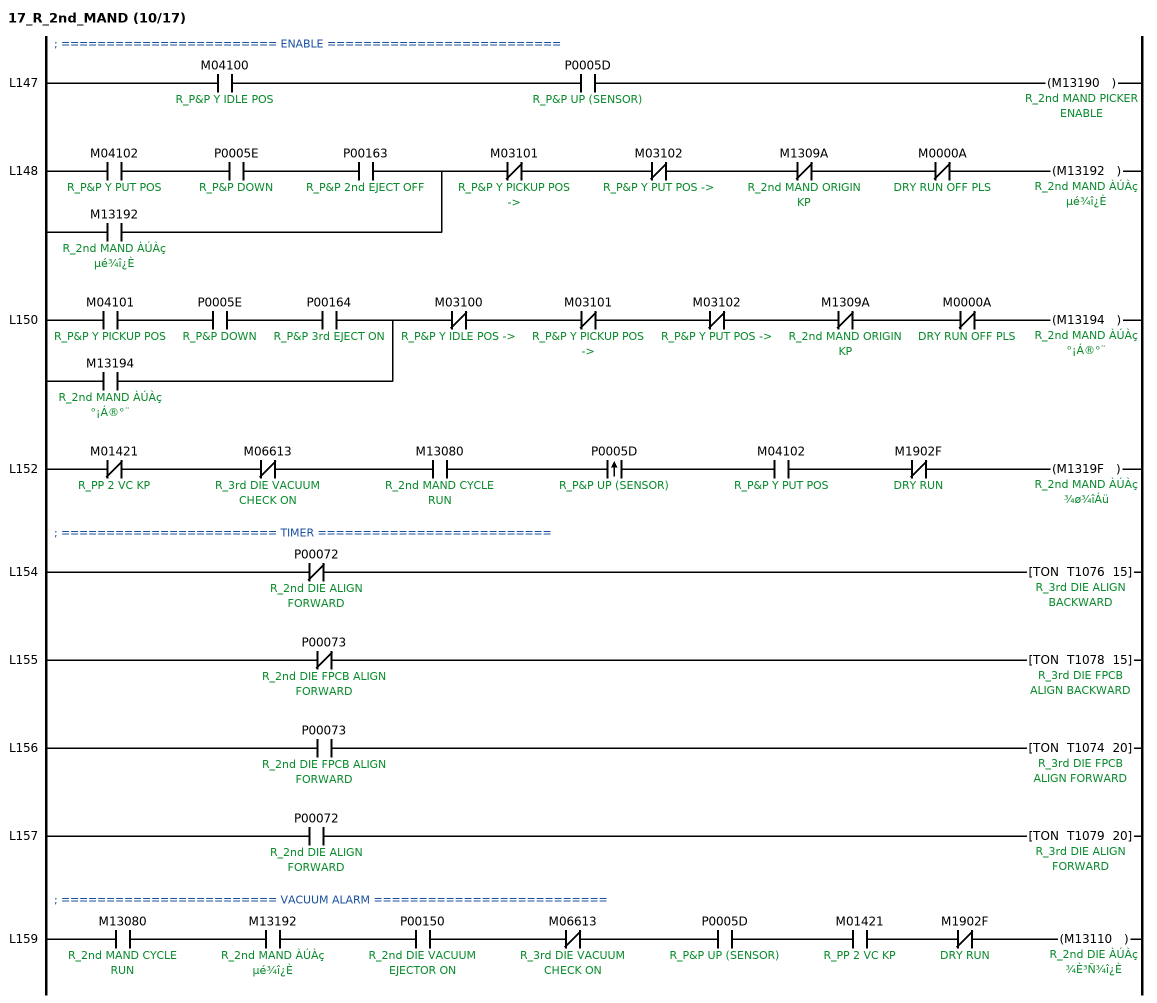
// ======================== ENABLE ==========================
; L147
LOAD      M04100	// R_P&P Y IDLE POS
AND       P0005D	// R_P&P UP (SENSOR)
OUT       M13190	// R_2nd MAND PICKER ENABLE
; L148
LOAD      M04102	// R_P&P Y PUT POS
AND       P0005E	// R_P&P DOWN
AND       P00163	// R_P&P 2nd EJECT OFF
OR        M13192	// R_2nd MAND ÀÚÀç µé¾î¿È
AND NOT   M03101	// R_P&P Y PICKUP POS ->
AND NOT   M03102	// R_P&P Y PUT POS ->
AND NOT   M1309A	// R_2nd MAND ORIGIN KP
AND NOT   M0000A	// DRY RUN OFF PLS
OUT       M13192	// R_2nd MAND ÀÚÀç µé¾î¿È
; L150
LOAD      M04101	// R_P&P Y PICKUP POS
AND       P0005E	// R_P&P DOWN
AND       P00164	// R_P&P 3rd EJECT ON
OR        M13194	// R_2nd MAND ÀÚÀç °¡Á®°¨
AND NOT   M03100	// R_P&P Y IDLE POS ->
AND NOT   M03101	// R_P&P Y PICKUP POS ->
AND NOT   M03102	// R_P&P Y PUT POS ->
AND NOT   M1309A	// R_2nd MAND ORIGIN KP
AND NOT   M0000A	// DRY RUN OFF PLS
OUT       M13194	// R_2nd MAND ÀÚÀç °¡Á®°¨
; L152
LOAD NOT  M01421	// R_PP 2 VC KP
AND NOT   M06613	// R_3rd DIE VACUUM CHECK ON
AND       M13080	// R_2nd MAND CYCLE RUN
ANDP      P0005D	// R_P&P UP (SENSOR)
AND       M04102	// R_P&P Y PUT POS
AND NOT   M1902F	// DRY RUN
OUT       M1319F	// R_2nd MAND ÀÚÀç ¾ø¾îÁü
// ======================== TIMER ==========================
; L154
LOAD NOT  P00072	// R_2nd DIE ALIGN FORWARD
TON       T1076 15	// R_3rd DIE ALIGN BACKWARD
; L155
LOAD NOT  P00073	// R_2nd DIE FPCB ALIGN FORWARD
TON       T1078 15	// R_3rd DIE FPCB ALIGN BACKWARD
; L156
LOAD      P00073	// R_2nd DIE FPCB ALIGN FORWARD
TON       T1074 20	// R_3rd DIE FPCB ALIGN FORWARD
; L157
LOAD      P00072	// R_2nd DIE ALIGN FORWARD
TON       T1079 20	// R_3rd DIE ALIGN FORWARD
// ======================== VACUUM ALARM ==========================
; L159
LOAD      M13080	// R_2nd MAND CYCLE RUN
AND       M13192	// R_2nd MAND ÀÚÀç µé¾î¿È
AND       P00150	// R_2nd DIE VACUUM EJECTOR ON
AND NOT   M06613	// R_3rd DIE VACUUM CHECK ON
AND       P0005D	// R_P&P UP (SENSOR)
AND       M01421	// R_PP 2 VC KP
AND NOT   M1902F	// DRY RUN
OUT       M13110	// R_2nd DIE ÀÚÀç ¾È³Ñ¾î¿È

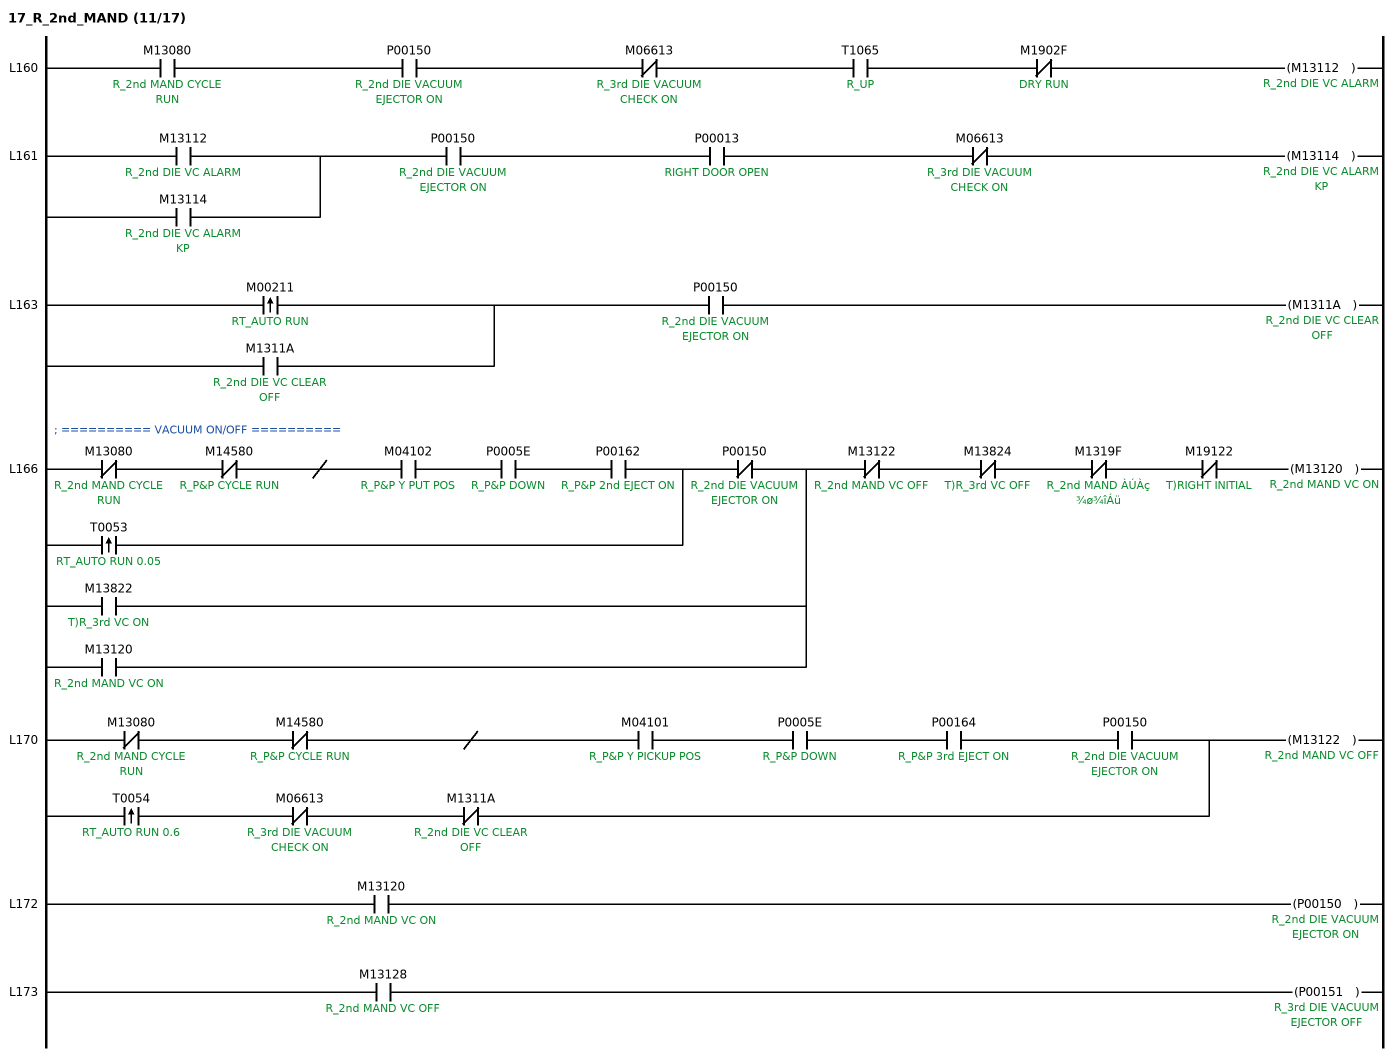
; L160
LOAD      M13080	// R_2nd MAND CYCLE RUN
AND       P00150	// R_2nd DIE VACUUM EJECTOR ON
AND NOT   M06613	// R_3rd DIE VACUUM CHECK ON
AND       T1065	// R_UP
AND NOT   M1902F	// DRY RUN
OUT       M13112	// R_2nd DIE VC ALARM
; L161
LOAD      M13112	// R_2nd DIE VC ALARM
OR        M13114	// R_2nd DIE VC ALARM KP
AND       P00150	// R_2nd DIE VACUUM EJECTOR ON
AND       P00013	// RIGHT DOOR OPEN
AND NOT   M06613	// R_3rd DIE VACUUM CHECK ON
OUT       M13114	// R_2nd DIE VC ALARM KP
; L163
LOADP     M00211	// RT_AUTO RUN
OR        M1311A	// R_2nd DIE VC CLEAR OFF
AND       P00150	// R_2nd DIE VACUUM EJECTOR ON
OUT       M1311A	// R_2nd DIE VC CLEAR OFF
// ========== VACUUM ON/OFF ==========
; L166
LOAD NOT  M13080	// R_2nd MAND CYCLE RUN
AND NOT   M14580	// R_P&P CYCLE RUN
NOT
AND       M04102	// R_P&P Y PUT POS
AND       P0005E	// R_P&P DOWN
AND       P00162	// R_P&P 2nd EJECT ON
ORP       T0053	// RT_AUTO RUN 0.05
AND NOT   P00150	// R_2nd DIE VACUUM EJECTOR ON
OR        M13822	// T)R_3rd VC ON
OR        M13120	// R_2nd MAND VC ON
AND NOT   M13122	// R_2nd MAND VC OFF
AND NOT   M13824	// T)R_3rd VC OFF
AND NOT   M1319F	// R_2nd MAND ÀÚÀç ¾ø¾îÁü
AND NOT   M19122	// T)RIGHT INITIAL
OUT       M13120	// R_2nd MAND VC ON
; L170
LOAD NOT  M13080	// R_2nd MAND CYCLE RUN
AND NOT   M14580	// R_P&P CYCLE RUN
NOT
AND       M04101	// R_P&P Y PICKUP POS
AND       P0005E	// R_P&P DOWN
AND       P00164	// R_P&P 3rd EJECT ON
AND       P00150	// R_2nd DIE VACUUM EJECTOR ON
LOADP     T0054	// RT_AUTO RUN 0.6
AND NOT   M06613	// R_3rd DIE VACUUM CHECK ON
AND NOT   M1311A	// R_2nd DIE VC CLEAR OFF
OR LOAD
OUT       M13122	// R_2nd MAND VC OFF
; L172
LOAD      M13120	// R_2nd MAND VC ON
OUT       P00150	// R_2nd DIE VACUUM EJECTOR ON
; L173
LOAD      M13128	// R_2nd MAND VC OFF
OUT       P00151	// R_3rd DIE VACUUM EJECTOR OFF

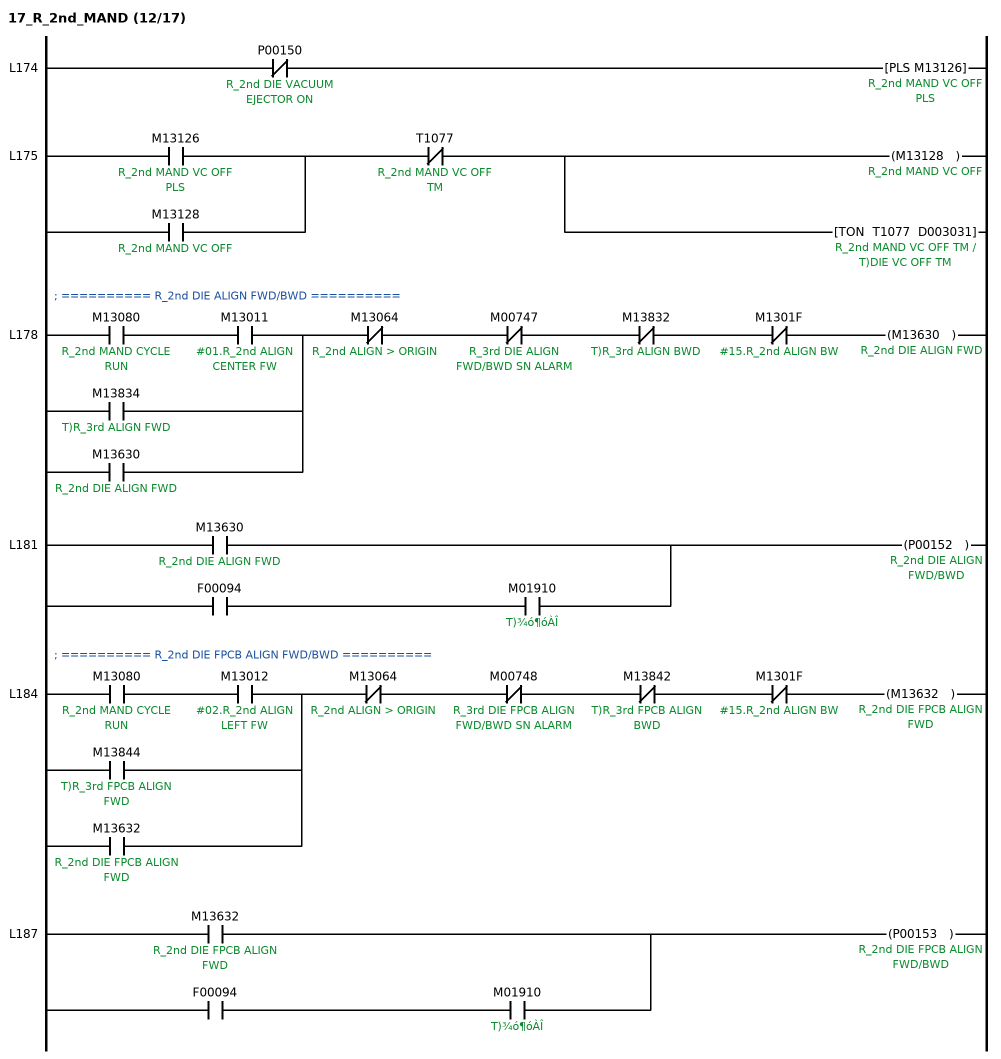
; L174
LOAD NOT  P00150	// R_2nd DIE VACUUM EJECTOR ON
OUTP      M13126	// R_2nd MAND VC OFF PLS
; L175
LOAD      M13126	// R_2nd MAND VC OFF PLS
OR        M13128	// R_2nd MAND VC OFF
AND NOT   T1077	// R_2nd MAND VC OFF TM
OUT       M13128	// R_2nd MAND VC OFF
TON       T1077 D003031	// R_2nd MAND VC OFF TM / T)DIE VC OFF TM
// ========== R_2nd DIE ALIGN FWD/BWD ==========
; L178
LOAD      M13080	// R_2nd MAND CYCLE RUN
AND       M13011	// #01.R_2nd ALIGN CENTER FW
OR        M13834	// T)R_3rd ALIGN FWD
OR        M13630	// R_2nd DIE ALIGN FWD
AND NOT   M13064	// R_2nd ALIGN > ORIGIN
AND NOT   M00747	// R_3rd DIE ALIGN FWD/BWD SN ALARM
AND NOT   M13832	// T)R_3rd ALIGN BWD
AND NOT   M1301F	// #15.R_2nd ALIGN BW
OUT       M13630	// R_2nd DIE ALIGN FWD
; L181
LOAD      M13630	// R_2nd DIE ALIGN FWD
LOAD      F00094
AND       M01910	// T)¾ó¶óÀÎ
OR LOAD
OUT       P00152	// R_2nd DIE ALIGN FWD/BWD
// ========== R_2nd DIE FPCB ALIGN FWD/BWD ==========
; L184
LOAD      M13080	// R_2nd MAND CYCLE RUN
AND       M13012	// #02.R_2nd ALIGN LEFT FW
OR        M13844	// T)R_3rd FPCB ALIGN FWD
OR        M13632	// R_2nd DIE FPCB ALIGN FWD
AND NOT   M13064	// R_2nd ALIGN > ORIGIN
AND NOT   M00748	// R_3rd DIE FPCB ALIGN FWD/BWD SN ALARM
AND NOT   M13842	// T)R_3rd FPCB ALIGN BWD
AND NOT   M1301F	// #15.R_2nd ALIGN BW
OUT       M13632	// R_2nd DIE FPCB ALIGN FWD
; L187
LOAD      M13632	// R_2nd DIE FPCB ALIGN FWD
LOAD      F00094
AND       M01910	// T)¾ó¶óÀÎ
OR LOAD
OUT       P00153	// R_2nd DIE FPCB ALIGN FWD/BWD

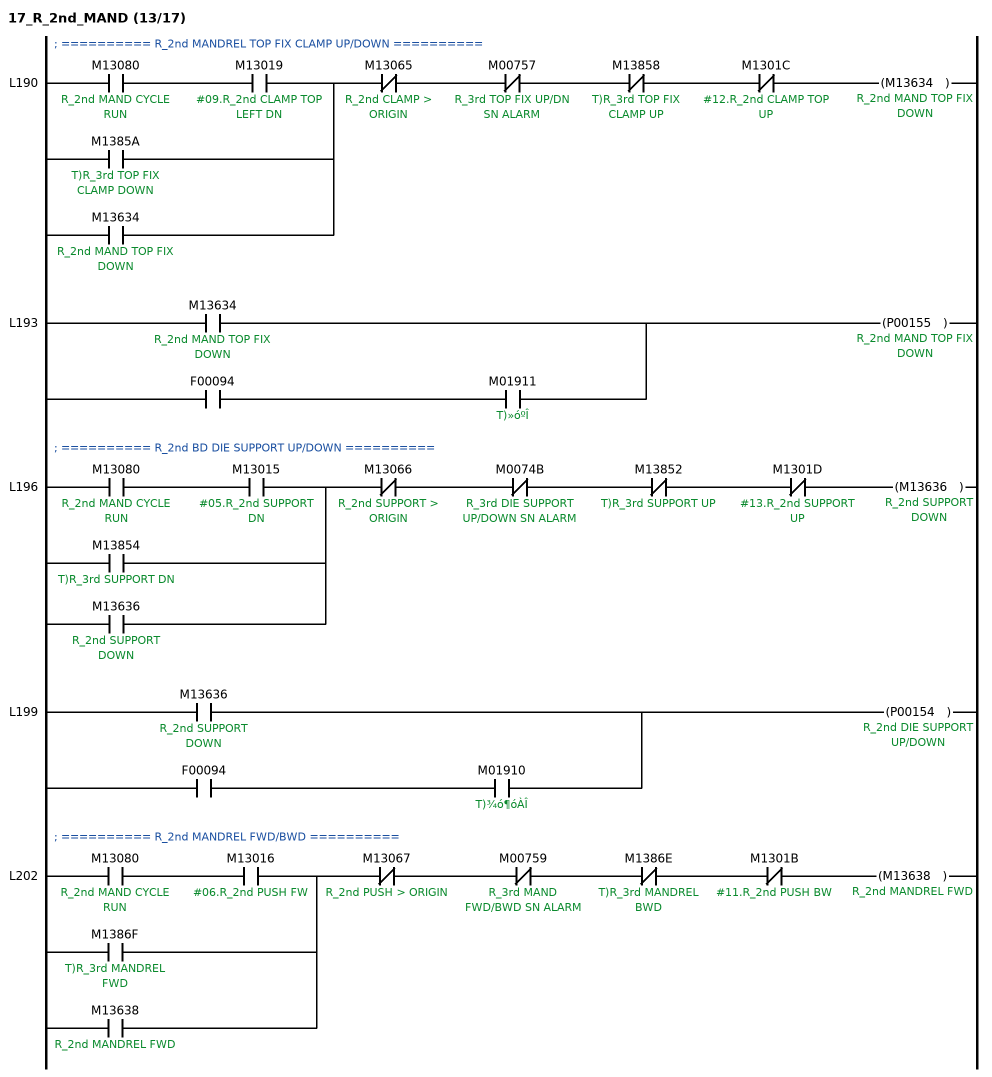
// ========== R_2nd MANDREL TOP FIX CLAMP UP/DOWN ==========
; L190
LOAD      M13080	// R_2nd MAND CYCLE RUN
AND       M13019	// #09.R_2nd CLAMP TOP LEFT DN
OR        M1385A	// T)R_3rd TOP FIX CLAMP DOWN
OR        M13634	// R_2nd MAND TOP FIX DOWN
AND NOT   M13065	// R_2nd CLAMP > ORIGIN
AND NOT   M00757	// R_3rd TOP FIX UP/DN SN ALARM
AND NOT   M13858	// T)R_3rd TOP FIX CLAMP UP
AND NOT   M1301C	// #12.R_2nd CLAMP TOP UP
OUT       M13634	// R_2nd MAND TOP FIX DOWN
; L193
LOAD      M13634	// R_2nd MAND TOP FIX DOWN
LOAD      F00094
AND       M01911	// T)»óºÎ
OR LOAD
OUT       P00155	// R_2nd MAND TOP FIX DOWN
// ========== R_2nd BD DIE SUPPORT UP/DOWN ==========
; L196
LOAD      M13080	// R_2nd MAND CYCLE RUN
AND       M13015	// #05.R_2nd SUPPORT DN
OR        M13854	// T)R_3rd SUPPORT DN
OR        M13636	// R_2nd SUPPORT DOWN
AND NOT   M13066	// R_2nd SUPPORT > ORIGIN
AND NOT   M0074B	// R_3rd DIE SUPPORT UP/DOWN SN ALARM
AND NOT   M13852	// T)R_3rd SUPPORT UP
AND NOT   M1301D	// #13.R_2nd SUPPORT UP
OUT       M13636	// R_2nd SUPPORT DOWN
; L199
LOAD      M13636	// R_2nd SUPPORT DOWN
LOAD      F00094
AND       M01910	// T)¾ó¶óÀÎ
OR LOAD
OUT       P00154	// R_2nd DIE SUPPORT UP/DOWN
// ========== R_2nd MANDREL FWD/BWD ==========
; L202
LOAD      M13080	// R_2nd MAND CYCLE RUN
AND       M13016	// #06.R_2nd PUSH FW
OR        M1386F	// T)R_3rd MANDREL FWD
OR        M13638	// R_2nd MANDREL FWD
AND NOT   M13067	// R_2nd PUSH > ORIGIN
AND NOT   M00759	// R_3rd MAND FWD/BWD SN ALARM
AND NOT   M1386E	// T)R_3rd MANDREL BWD
AND NOT   M1301B	// #11.R_2nd PUSH BW
OUT       M13638	// R_2nd MANDREL FWD

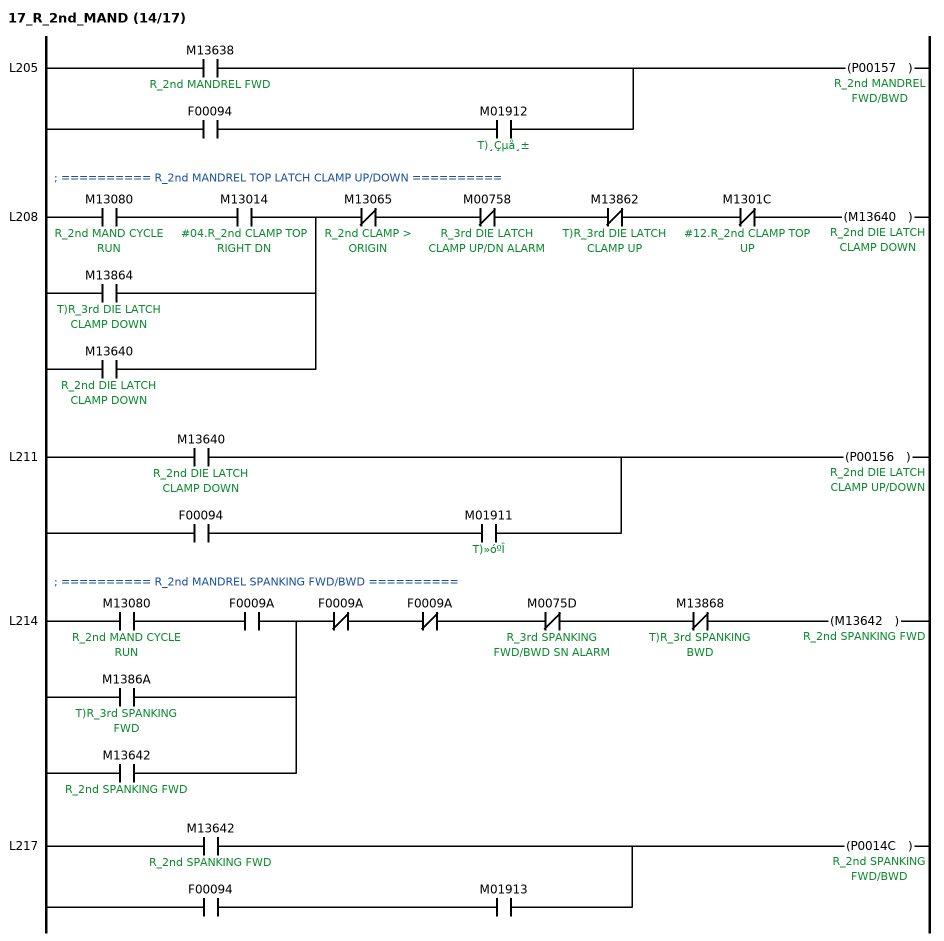
; L205
LOAD      M13638	// R_2nd MANDREL FWD
LOAD      F00094
AND       M01912	// T)¸Çµå¸±
OR LOAD
OUT       P00157	// R_2nd MANDREL FWD/BWD
// ========== R_2nd MANDREL TOP LATCH CLAMP UP/DOWN ==========
; L208
LOAD      M13080	// R_2nd MAND CYCLE RUN
AND       M13014	// #04.R_2nd CLAMP TOP RIGHT DN
OR        M13864	// T)R_3rd DIE LATCH CLAMP DOWN
OR        M13640	// R_2nd DIE LATCH CLAMP DOWN
AND NOT   M13065	// R_2nd CLAMP > ORIGIN
AND NOT   M00758	// R_3rd DIE LATCH CLAMP UP/DN ALARM
AND NOT   M13862	// T)R_3rd DIE LATCH CLAMP UP
AND NOT   M1301C	// #12.R_2nd CLAMP TOP UP
OUT       M13640	// R_2nd DIE LATCH CLAMP DOWN
; L211
LOAD      M13640	// R_2nd DIE LATCH CLAMP DOWN
LOAD      F00094
AND       M01911	// T)»óºÎ
OR LOAD
OUT       P00156	// R_2nd DIE LATCH CLAMP UP/DOWN
// ========== R_2nd MANDREL SPANKING FWD/BWD ==========
; L214
LOAD      M13080	// R_2nd MAND CYCLE RUN
AND       F0009A
OR        M1386A	// T)R_3rd SPANKING FWD
OR        M13642	// R_2nd SPANKING FWD
AND NOT   F0009A
AND NOT   F0009A
AND NOT   M0075D	// R_3rd SPANKING FWD/BWD SN ALARM
AND NOT   M13868	// T)R_3rd SPANKING BWD
OUT       M13642	// R_2nd SPANKING FWD
; L217
LOAD      M13642	// R_2nd SPANKING FWD
LOAD      F00094
AND       M01913
OR LOAD
OUT       P0014C	// R_2nd SPANKING FWD/BWD

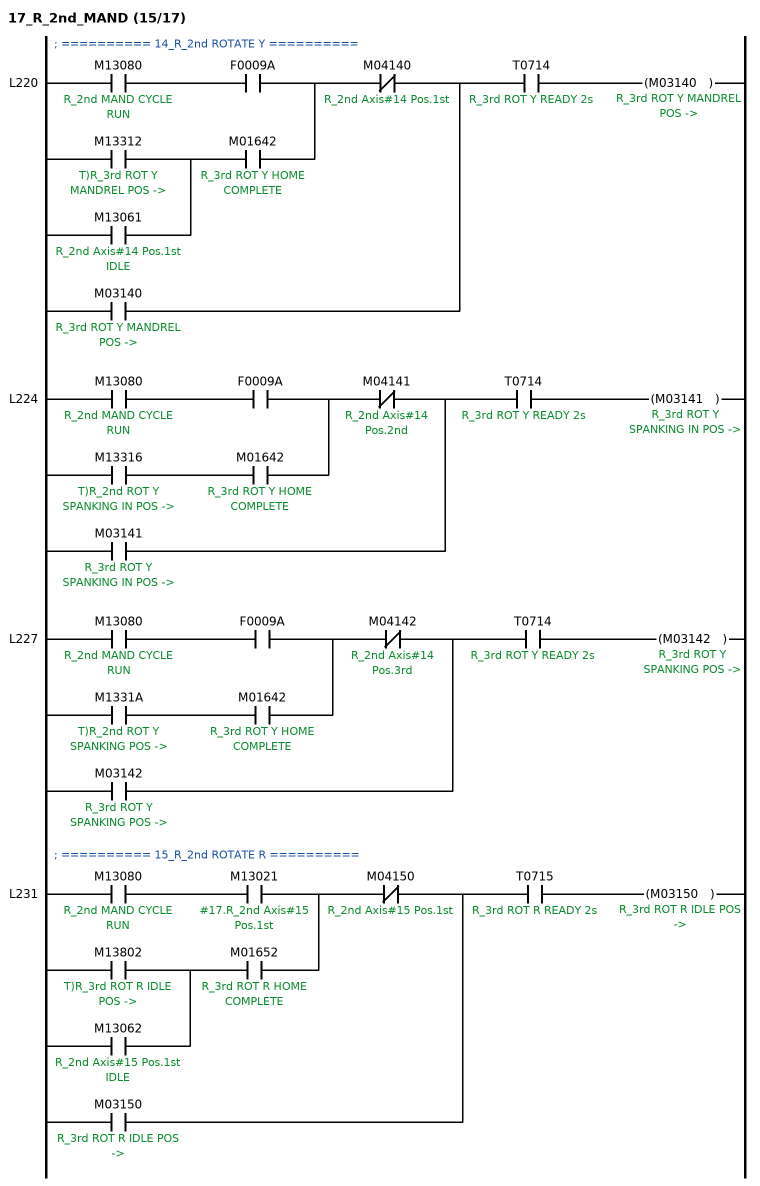
// ========== 14_R_2nd ROTATE Y ==========
; L220
LOAD      M13080	// R_2nd MAND CYCLE RUN
AND       F0009A
LOAD      M13312	// T)R_3rd ROT Y MANDREL POS ->
OR        M13061	// R_2nd Axis#14 Pos.1st IDLE
AND       M01642	// R_3rd ROT Y HOME COMPLETE
OR LOAD
AND NOT   M04140	// R_2nd Axis#14 Pos.1st
OR        M03140	// R_3rd ROT Y MANDREL POS ->
AND       T0714	// R_3rd ROT Y READY 2s
OUT       M03140	// R_3rd ROT Y MANDREL POS ->
; L224
LOAD      M13080	// R_2nd MAND CYCLE RUN
AND       F0009A
LOAD      M13316	// T)R_2nd ROT Y SPANKING IN POS ->
AND       M01642	// R_3rd ROT Y HOME COMPLETE
OR LOAD
AND NOT   M04141	// R_2nd Axis#14 Pos.2nd
OR        M03141	// R_3rd ROT Y SPANKING IN POS ->
AND       T0714	// R_3rd ROT Y READY 2s
OUT       M03141	// R_3rd ROT Y SPANKING IN POS ->
; L227
LOAD      M13080	// R_2nd MAND CYCLE RUN
AND       F0009A
LOAD      M1331A	// T)R_2nd ROT Y SPANKING POS ->
AND       M01642	// R_3rd ROT Y HOME COMPLETE
OR LOAD
AND NOT   M04142	// R_2nd Axis#14 Pos.3rd
OR        M03142	// R_3rd ROT Y SPANKING POS ->
AND       T0714	// R_3rd ROT Y READY 2s
OUT       M03142	// R_3rd ROT Y SPANKING POS ->
// ========== 15_R_2nd ROTATE R ==========
; L231
LOAD      M13080	// R_2nd MAND CYCLE RUN
AND       M13021	// #17.R_2nd Axis#15 Pos.1st
LOAD      M13802	// T)R_3rd ROT R IDLE POS ->
OR        M13062	// R_2nd Axis#15 Pos.1st IDLE
AND       M01652	// R_3rd ROT R HOME COMPLETE
OR LOAD
AND NOT   M04150	// R_2nd Axis#15 Pos.1st
OR        M03150	// R_3rd ROT R IDLE POS ->
AND       T0715	// R_3rd ROT R READY 2s
OUT       M03150	// R_3rd ROT R IDLE POS ->

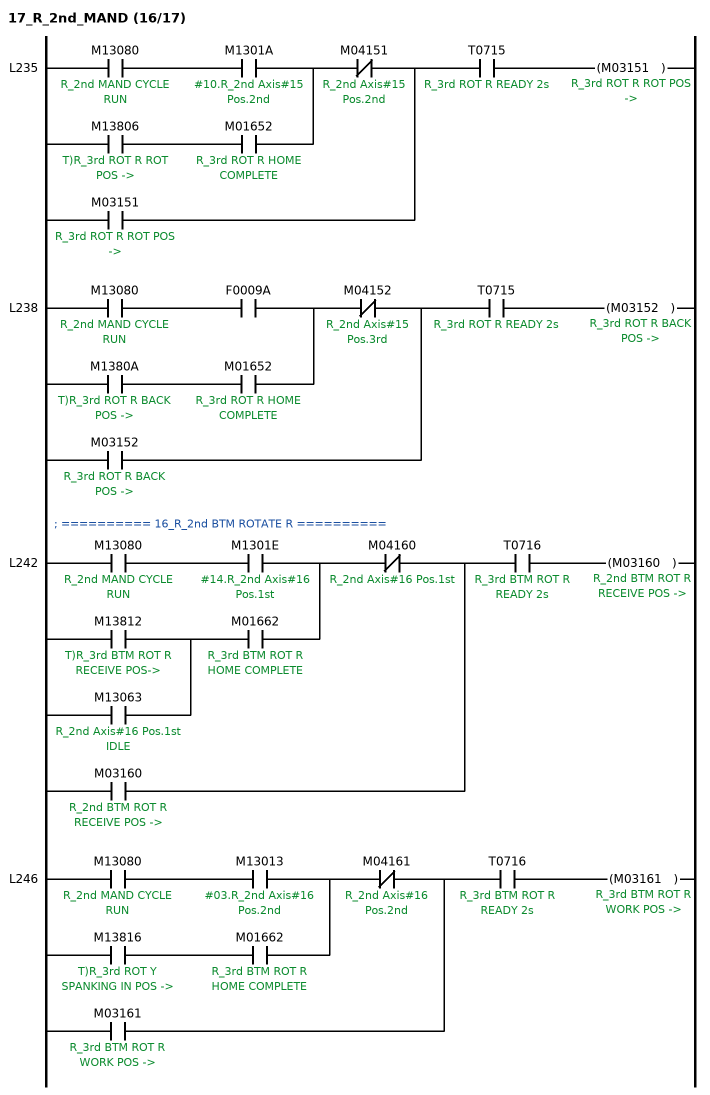
; L235
LOAD      M13080	// R_2nd MAND CYCLE RUN
AND       M1301A	// #10.R_2nd Axis#15 Pos.2nd
LOAD      M13806	// T)R_3rd ROT R ROT POS ->
AND       M01652	// R_3rd ROT R HOME COMPLETE
OR LOAD
AND NOT   M04151	// R_2nd Axis#15 Pos.2nd
OR        M03151	// R_3rd ROT R ROT POS ->
AND       T0715	// R_3rd ROT R READY 2s
OUT       M03151	// R_3rd ROT R ROT POS ->
; L238
LOAD      M13080	// R_2nd MAND CYCLE RUN
AND       F0009A
LOAD      M1380A	// T)R_3rd ROT R BACK POS ->
AND       M01652	// R_3rd ROT R HOME COMPLETE
OR LOAD
AND NOT   M04152	// R_2nd Axis#15 Pos.3rd
OR        M03152	// R_3rd ROT R BACK POS ->
AND       T0715	// R_3rd ROT R READY 2s
OUT       M03152	// R_3rd ROT R BACK POS ->
// ========== 16_R_2nd BTM ROTATE R ==========
; L242
LOAD      M13080	// R_2nd MAND CYCLE RUN
AND       M1301E	// #14.R_2nd Axis#16 Pos.1st
LOAD      M13812	// T)R_3rd BTM ROT R RECEIVE POS->
OR        M13063	// R_2nd Axis#16 Pos.1st IDLE
AND       M01662	// R_3rd BTM ROT R HOME COMPLETE
OR LOAD
AND NOT   M04160	// R_2nd Axis#16 Pos.1st
OR        M03160	// R_2nd BTM ROT R RECEIVE POS ->
AND       T0716	// R_3rd BTM ROT R READY 2s
OUT       M03160	// R_2nd BTM ROT R RECEIVE POS ->
; L246
LOAD      M13080	// R_2nd MAND CYCLE RUN
AND       M13013	// #03.R_2nd Axis#16 Pos.2nd
LOAD      M13816	// T)R_3rd ROT Y SPANKING IN POS ->
AND       M01662	// R_3rd BTM ROT R HOME COMPLETE
OR LOAD
AND NOT   M04161	// R_2nd Axis#16 Pos.2nd
OR        M03161	// R_3rd BTM ROT R WORK POS ->
AND       T0716	// R_3rd BTM ROT R READY 2s
OUT       M03161	// R_3rd BTM ROT R WORK POS ->

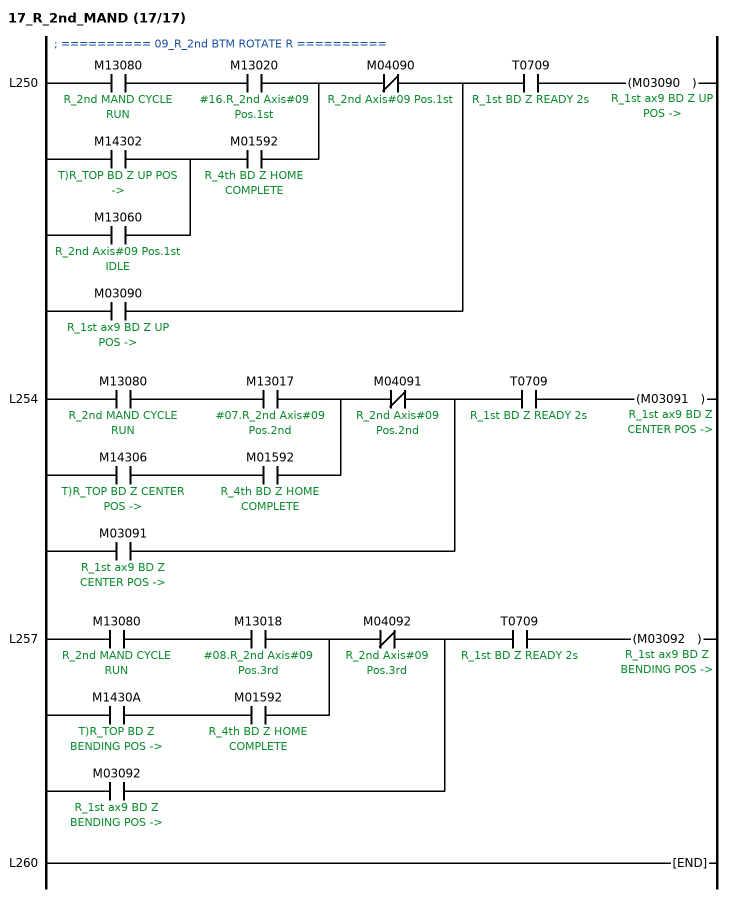
// ========== 09_R_2nd BTM ROTATE R ==========
; L250
LOAD      M13080	// R_2nd MAND CYCLE RUN
AND       M13020	// #16.R_2nd Axis#09 Pos.1st
LOAD      M14302	// T)R_TOP BD Z UP POS ->
OR        M13060	// R_2nd Axis#09 Pos.1st IDLE
AND       M01592	// R_4th BD Z HOME COMPLETE
OR LOAD
AND NOT   M04090	// R_2nd Axis#09 Pos.1st
OR        M03090	// R_1st ax9 BD Z UP POS ->
AND       T0709	// R_1st BD Z READY 2s
OUT       M03090	// R_1st ax9 BD Z UP POS ->
; L254
LOAD      M13080	// R_2nd MAND CYCLE RUN
AND       M13017	// #07.R_2nd Axis#09 Pos.2nd
LOAD      M14306	// T)R_TOP BD Z CENTER POS ->
AND       M01592	// R_4th BD Z HOME COMPLETE
OR LOAD
AND NOT   M04091	// R_2nd Axis#09 Pos.2nd
OR        M03091	// R_1st ax9 BD Z CENTER POS ->
AND       T0709	// R_1st BD Z READY 2s
OUT       M03091	// R_1st ax9 BD Z CENTER POS ->
; L257
LOAD      M13080	// R_2nd MAND CYCLE RUN
AND       M13018	// #08.R_2nd Axis#09 Pos.3rd
LOAD      M1430A	// T)R_TOP BD Z BENDING POS ->
AND       M01592	// R_4th BD Z HOME COMPLETE
OR LOAD
AND NOT   M04092	// R_2nd Axis#09 Pos.3rd
OR        M03092	// R_1st ax9 BD Z BENDING POS ->
AND       T0709	// R_1st BD Z READY 2s
OUT       M03092	// R_1st ax9 BD Z BENDING POS ->
; L260
END

PROGRAM 18_R_3rd_MAND (task: ½ºÄµ ÇÁ·Î±×·¥)

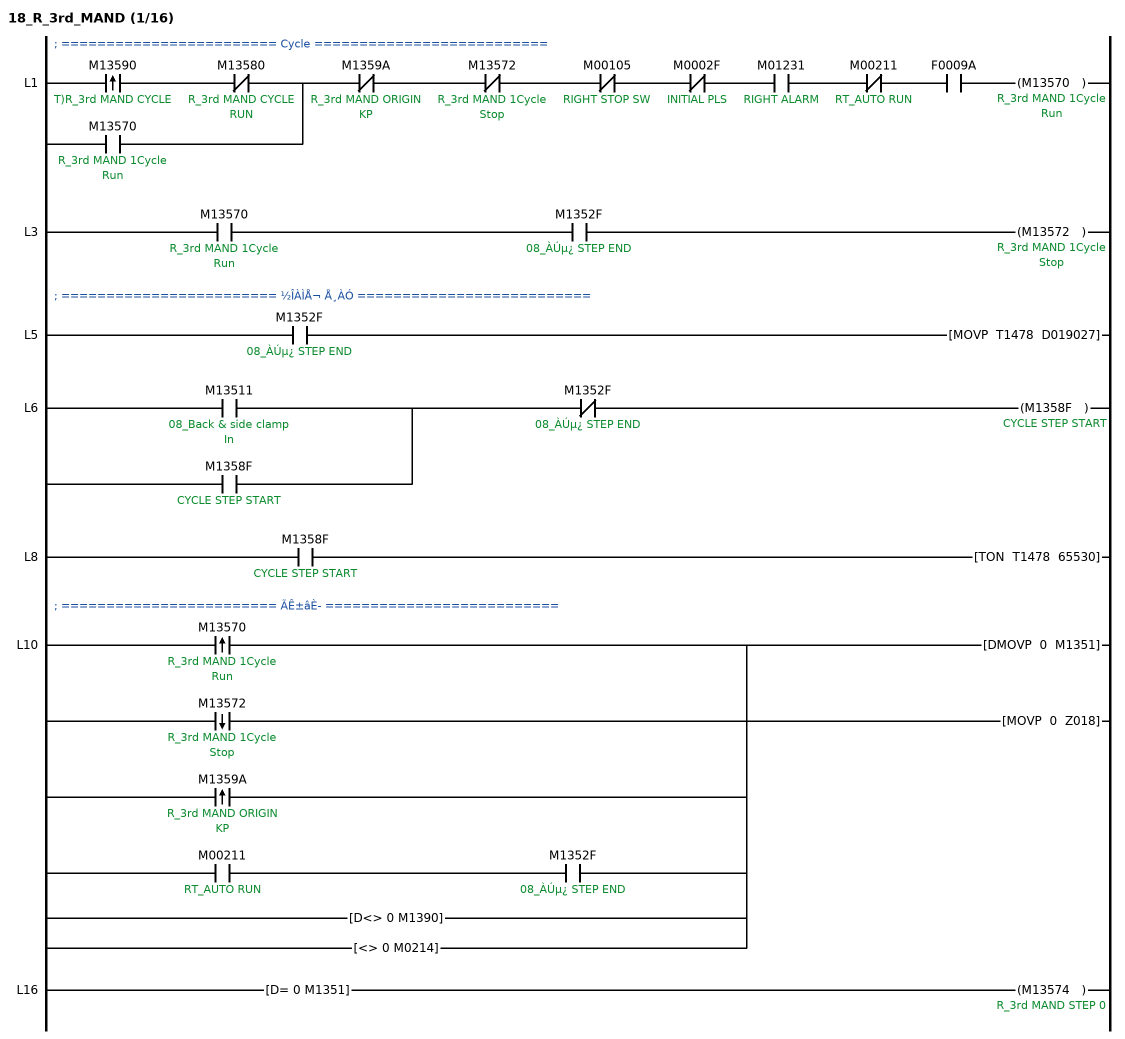
// ======================== Cycle ==========================
; L1
LOADP     M13590	// T)R_3rd MAND CYCLE
AND NOT   M13580	// R_3rd MAND CYCLE RUN
OR        M13570	// R_3rd MAND 1Cycle Run
AND NOT   M1359A	// R_3rd MAND ORIGIN KP
AND NOT   M13572	// R_3rd MAND 1Cycle Stop
AND NOT   M00105	// RIGHT STOP SW
AND NOT   M0002F	// INITIAL PLS
AND       M01231	// RIGHT ALARM
AND NOT   M00211	// RT_AUTO RUN
AND       F0009A
OUT       M13570	// R_3rd MAND 1Cycle Run
; L3
LOAD      M13570	// R_3rd MAND 1Cycle Run
AND       M1352F	// 08_ÀÚµ¿ STEP END
OUT       M13572	// R_3rd MAND 1Cycle Stop
// ======================== ½ÎÀÌÅ¬ Å¸ÀÓ ==========================
; L5
LOAD      M1352F	// 08_ÀÚµ¿ STEP END
MOVP      T1478 D019027
; L6
LOAD      M13511	// 08_Back & side clamp In
OR        M1358F	// CYCLE STEP START
AND NOT   M1352F	// 08_ÀÚµ¿ STEP END
OUT       M1358F	// CYCLE STEP START
; L8
LOAD      M1358F	// CYCLE STEP START
TON       T1478 65530
// ======================== ÃÊ±âÈ­ ==========================
; L10
LOADP     M13570	// R_3rd MAND 1Cycle Run
ORN       M13572	// R_3rd MAND 1Cycle Stop
ORP       M1359A	// R_3rd MAND ORIGIN KP
LOAD      M00211	// RT_AUTO RUN
AND       M1352F	// 08_ÀÚµ¿ STEP END
OR LOAD
ORD<>     0 M1390
OR<>      0 M0214
DMOVP     0 M1351
MOVP      0 Z018
; L16
LOADD=    0 M1351
OUT       M13574	// R_3rd MAND STEP 0

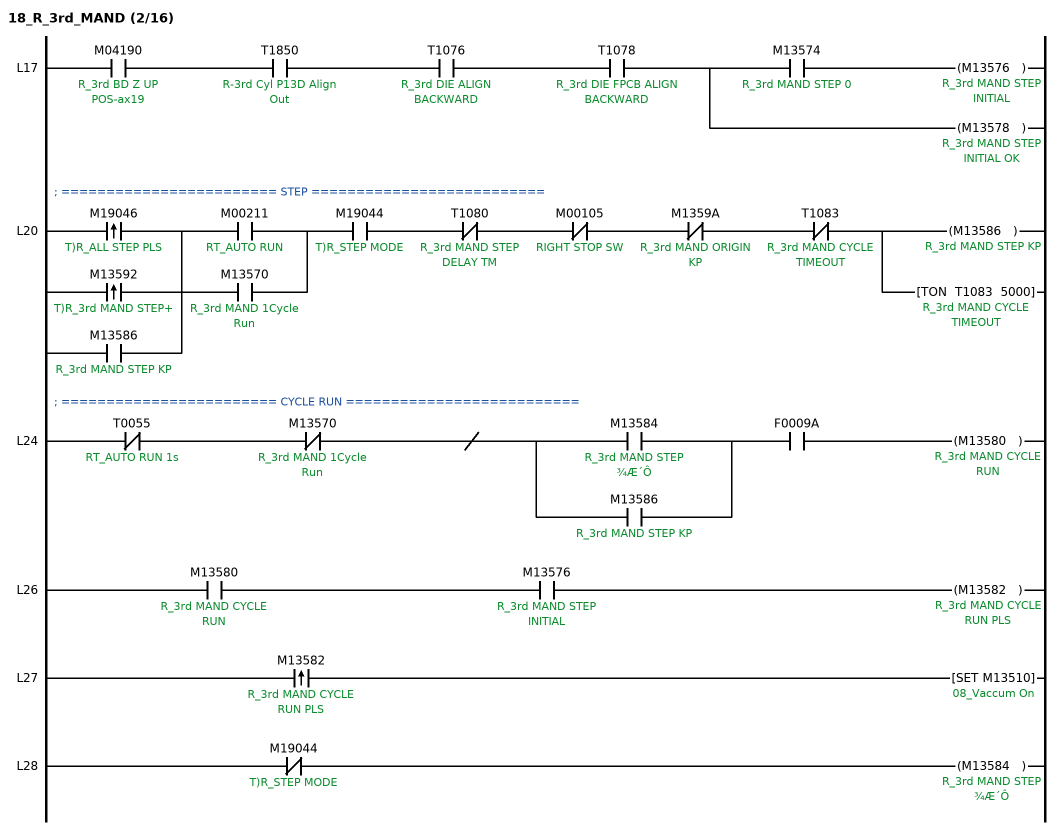
; L17
LOAD      M04190	// R_3rd BD Z UP POS-ax19
AND       T1850	// R-3rd Cyl P13D Align Out
AND       T1076	// R_3rd DIE ALIGN BACKWARD
AND       T1078	// R_3rd DIE FPCB ALIGN BACKWARD
MPUSH
AND       M13574	// R_3rd MAND STEP 0
OUT       M13576	// R_3rd MAND STEP INITIAL
MPOP
OUT       M13578	// R_3rd MAND STEP INITIAL OK
// ======================== STEP ==========================
; L20
LOADP     M19046	// T)R_ALL STEP PLS
ORP       M13592	// T)R_3rd MAND STEP+
OR        M13586	// R_3rd MAND STEP KP
LOAD      M00211	// RT_AUTO RUN
OR        M13570	// R_3rd MAND 1Cycle Run
AND LOAD
AND       M19044	// T)R_STEP MODE
AND NOT   T1080	// R_3rd MAND STEP DELAY TM
AND NOT   M00105	// RIGHT STOP SW
AND NOT   M1359A	// R_3rd MAND ORIGIN KP
AND NOT   T1083	// R_3rd MAND CYCLE TIMEOUT
OUT       M13586	// R_3rd MAND STEP KP
TON       T1083 5000	// R_3rd MAND CYCLE TIMEOUT
// ======================== CYCLE RUN ==========================
; L24
LOAD NOT  T0055	// RT_AUTO RUN 1s
AND NOT   M13570	// R_3rd MAND 1Cycle Run
NOT
LOAD      M13584	// R_3rd MAND STEP ¾Æ´Ô
OR        M13586	// R_3rd MAND STEP KP
AND LOAD
AND       F0009A
OUT       M13580	// R_3rd MAND CYCLE RUN
; L26
LOAD      M13580	// R_3rd MAND CYCLE RUN
AND       M13576	// R_3rd MAND STEP INITIAL
OUT       M13582	// R_3rd MAND CYCLE RUN PLS
; L27
LOADP     M13582	// R_3rd MAND CYCLE RUN PLS
SET       M13510	// 08_Vaccum On
; L28
LOAD NOT  M19044	// T)R_STEP MODE
OUT       M13584	// R_3rd MAND STEP ¾Æ´Ô

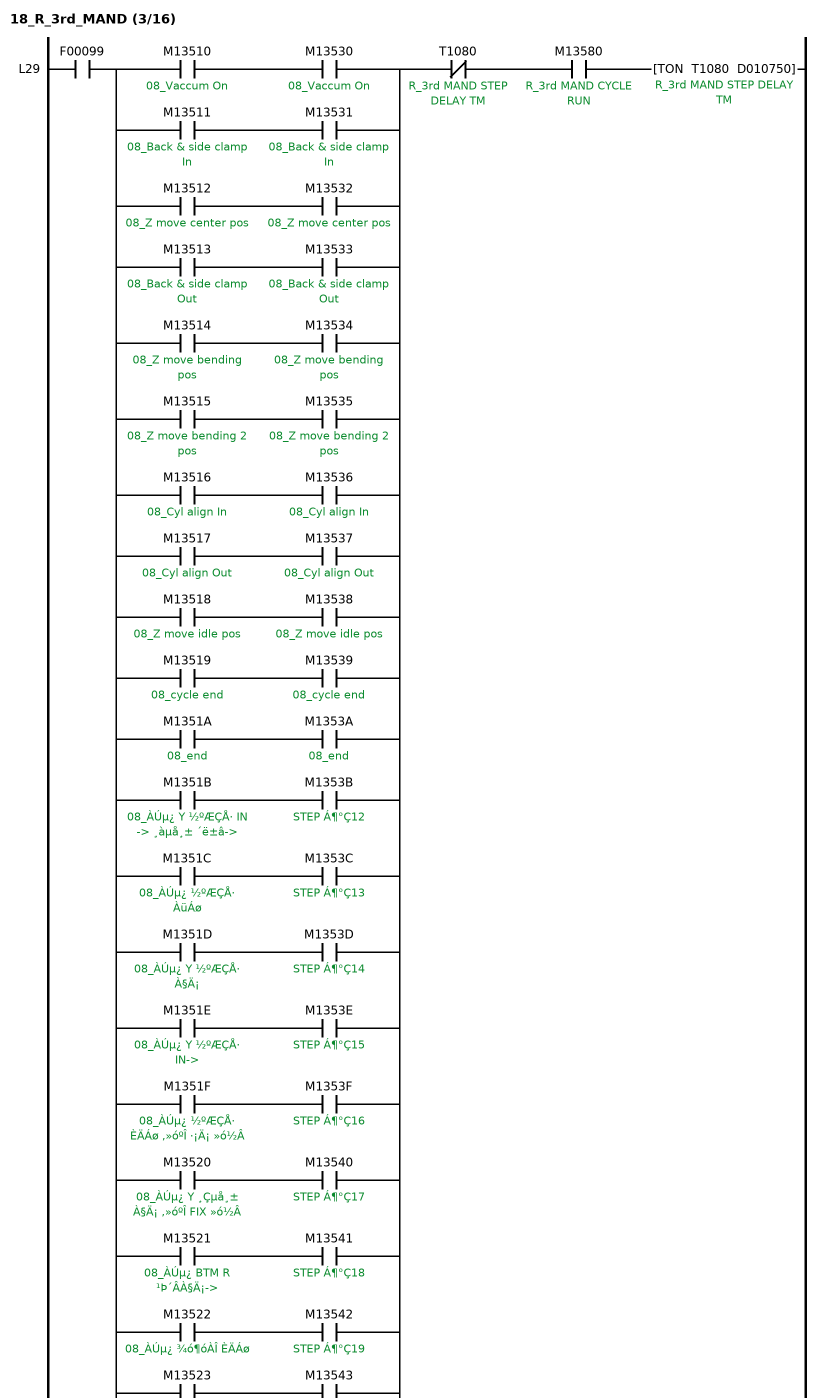

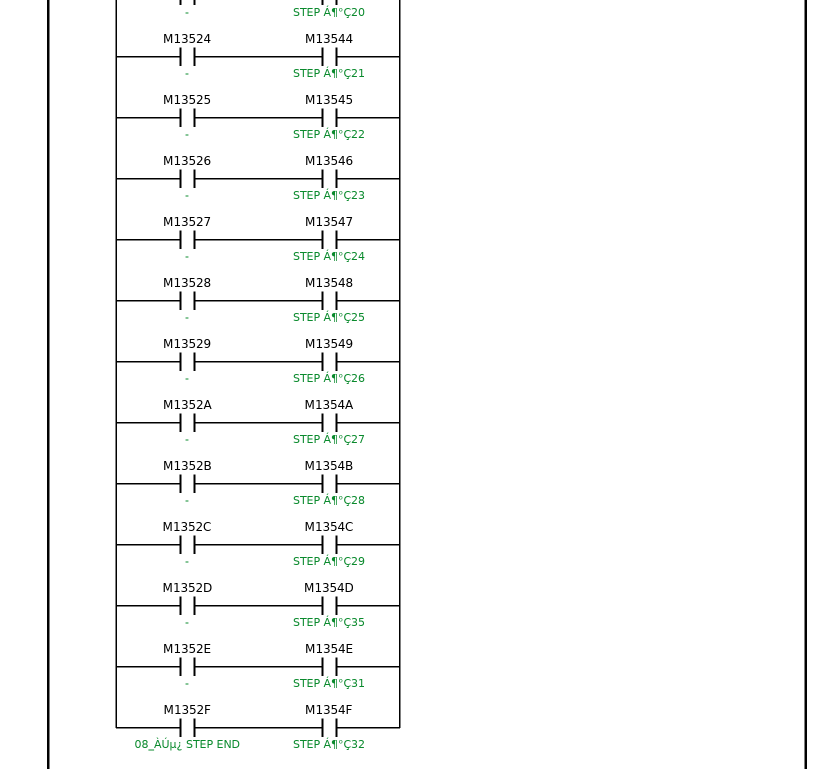
; L29
LOAD      F00099
LOAD      M13510	// 08_Vaccum On
AND       M13530	// 08_Vaccum On
LOAD      M13511	// 08_Back & side clamp In
AND       M13531	// 08_Back & side clamp In
OR LOAD
LOAD      M13512	// 08_Z move center pos
AND       M13532	// 08_Z move center pos
OR LOAD
LOAD      M13513	// 08_Back & side clamp Out
AND       M13533	// 08_Back & side clamp Out
OR LOAD
LOAD      M13514	// 08_Z move bending pos
AND       M13534	// 08_Z move bending pos
OR LOAD
LOAD      M13515	// 08_Z move bending 2 pos
AND       M13535	// 08_Z move bending 2 pos
OR LOAD
LOAD      M13516	// 08_Cyl align In
AND       M13536	// 08_Cyl align In
OR LOAD
LOAD      M13517	// 08_Cyl align Out
AND       M13537	// 08_Cyl align Out
OR LOAD
LOAD      M13518	// 08_Z move idle pos
AND       M13538	// 08_Z move idle pos
OR LOAD
LOAD      M13519	// 08_cycle end
AND       M13539	// 08_cycle end
OR LOAD
LOAD      M1351A	// 08_end
AND       M1353A	// 08_end
OR LOAD
LOAD      M1351B	// 08_ÀÚµ¿ Y ½ºÆÇÅ· IN -> ¸àµå¸± ´ë±â->
AND       M1353B	// STEP Á¶°Ç12
OR LOAD
LOAD      M1351C	// 08_ÀÚµ¿ ½ºÆÇÅ· ÀüÁø
AND       M1353C	// STEP Á¶°Ç13
OR LOAD
LOAD      M1351D	// 08_ÀÚµ¿ Y ½ºÆÇÅ· À§Ä¡
AND       M1353D	// STEP Á¶°Ç14
OR LOAD
LOAD      M1351E	// 08_ÀÚµ¿ Y ½ºÆÇÅ· IN->
AND       M1353E	// STEP Á¶°Ç15
OR LOAD
LOAD      M1351F	// 08_ÀÚµ¿ ½ºÆÇÅ· ÈÄÁø ,»óºÎ ·¡Ä¡ »ó½Â
AND       M1353F	// STEP Á¶°Ç16
OR LOAD
LOAD      M13520	// 08_ÀÚµ¿ Y ¸Çµå¸± À§Ä¡ ,»óºÎ FIX »ó½Â
AND       M13540	// STEP Á¶°Ç17
OR LOAD
LOAD      M13521	// 08_ÀÚµ¿ BTM R ¹Þ´ÂÀ§Ä¡->
AND       M13541	// STEP Á¶°Ç18
OR LOAD
LOAD      M13522	// 08_ÀÚµ¿ ¾ó¶óÀÎ ÈÄÁø
AND       M13542	// STEP Á¶°Ç19
OR LOAD
LOAD      M13523	// -
AND       M13543	// STEP Á¶°Ç20
OR LOAD
LOAD      M13524	// -
AND       M13544	// STEP Á¶°Ç21
OR LOAD
LOAD      M13525	// -
AND       M13545	// STEP Á¶°Ç22
OR LOAD
LOAD      M13526	// -
AND       M13546	// STEP Á¶°Ç23
OR LOAD
LOAD      M13527	// -
AND       M13547	// STEP Á¶°Ç24
OR LOAD
LOAD      M13528	// -
AND       M13548	// STEP Á¶°Ç25
OR LOAD
LOAD      M13529	// -
AND       M13549	// STEP Á¶°Ç26
OR LOAD
LOAD      M1352A	// -
AND       M1354A	// STEP Á¶°Ç27
OR LOAD
LOAD      M1352B	// -
AND       M1354B	// STEP Á¶°Ç28
OR LOAD
LOAD      M1352C	// -
AND       M1354C	// STEP Á¶°Ç29
OR LOAD
LOAD      M1352D	// -
AND       M1354D	// STEP Á¶°Ç35
OR LOAD
LOAD      M1352E	// -
AND       M1354E	// STEP Á¶°Ç31
OR LOAD
LOAD      M1352F	// 08_ÀÚµ¿ STEP END
AND       M1354F	// STEP Á¶°Ç32
OR LOAD
AND LOAD
AND NOT   T1080	// R_3rd MAND STEP DELAY TM
AND       M13580	// R_3rd MAND CYCLE RUN
TON       T1080 D010750	// R_3rd MAND STEP DELAY TM

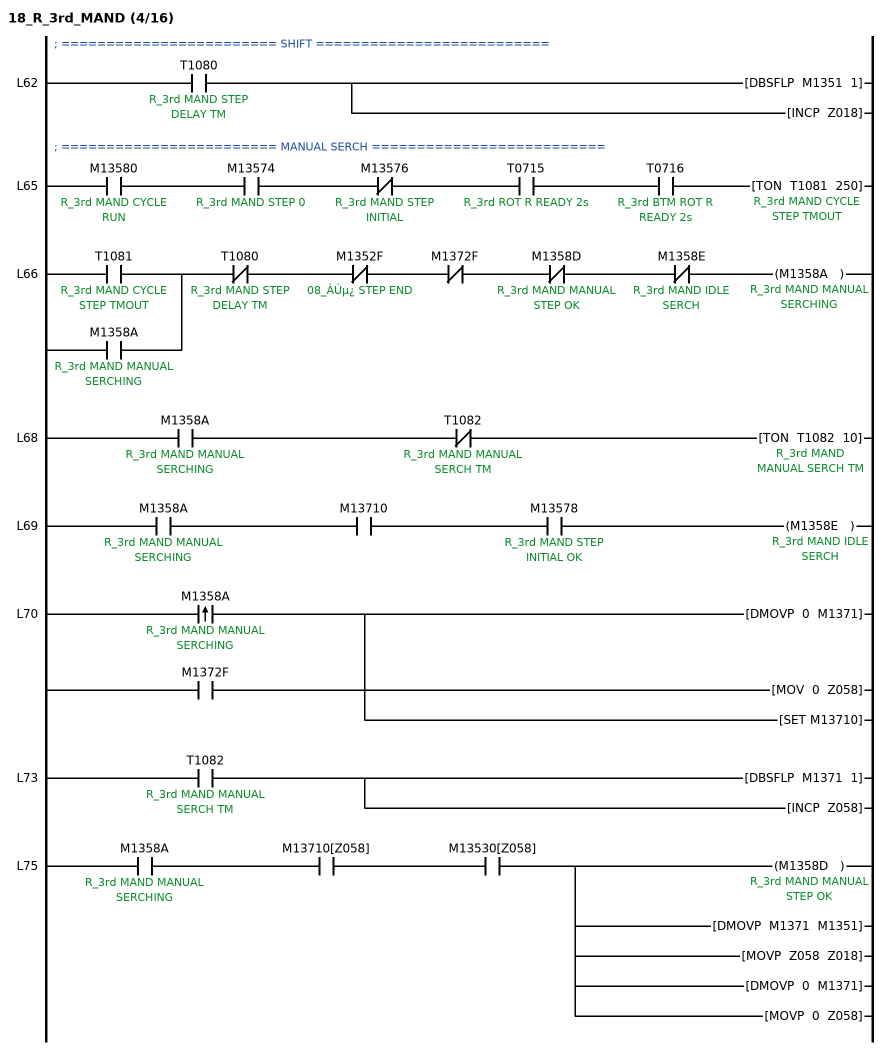
// ======================== SHIFT ==========================
; L62
LOAD      T1080	// R_3rd MAND STEP DELAY TM
DBSFLP    M1351 1
INCP      Z018
// ======================== MANUAL SERCH ==========================
; L65
LOAD      M13580	// R_3rd MAND CYCLE RUN
AND       M13574	// R_3rd MAND STEP 0
AND NOT   M13576	// R_3rd MAND STEP INITIAL
AND       T0715	// R_3rd ROT R READY 2s
AND       T0716	// R_3rd BTM ROT R READY 2s
TON       T1081 250	// R_3rd MAND CYCLE STEP TMOUT
; L66
LOAD      T1081	// R_3rd MAND CYCLE STEP TMOUT
OR        M1358A	// R_3rd MAND MANUAL SERCHING
AND NOT   T1080	// R_3rd MAND STEP DELAY TM
AND NOT   M1352F	// 08_ÀÚµ¿ STEP END
AND NOT   M1372F
AND NOT   M1358D	// R_3rd MAND MANUAL STEP OK
AND NOT   M1358E	// R_3rd MAND IDLE SERCH
OUT       M1358A	// R_3rd MAND MANUAL SERCHING
; L68
LOAD      M1358A	// R_3rd MAND MANUAL SERCHING
AND NOT   T1082	// R_3rd MAND MANUAL SERCH TM
TON       T1082 10	// R_3rd MAND MANUAL SERCH TM
; L69
LOAD      M1358A	// R_3rd MAND MANUAL SERCHING
AND       M13710
AND       M13578	// R_3rd MAND STEP INITIAL OK
OUT       M1358E	// R_3rd MAND IDLE SERCH
; L70
LOADP     M1358A	// R_3rd MAND MANUAL SERCHING
OR        M1372F
DMOVP     0 M1371
MOV       0 Z058
SET       M13710
; L73
LOAD      T1082	// R_3rd MAND MANUAL SERCH TM
DBSFLP    M1371 1
INCP      Z058
; L75
LOAD      M1358A	// R_3rd MAND MANUAL SERCHING
AND       M13710[Z058]
AND       M13530[Z058]
OUT       M1358D	// R_3rd MAND MANUAL STEP OK
DMOVP     M1371 M1351
MOVP      Z058 Z018
DMOVP     0 M1371
MOVP      0 Z058

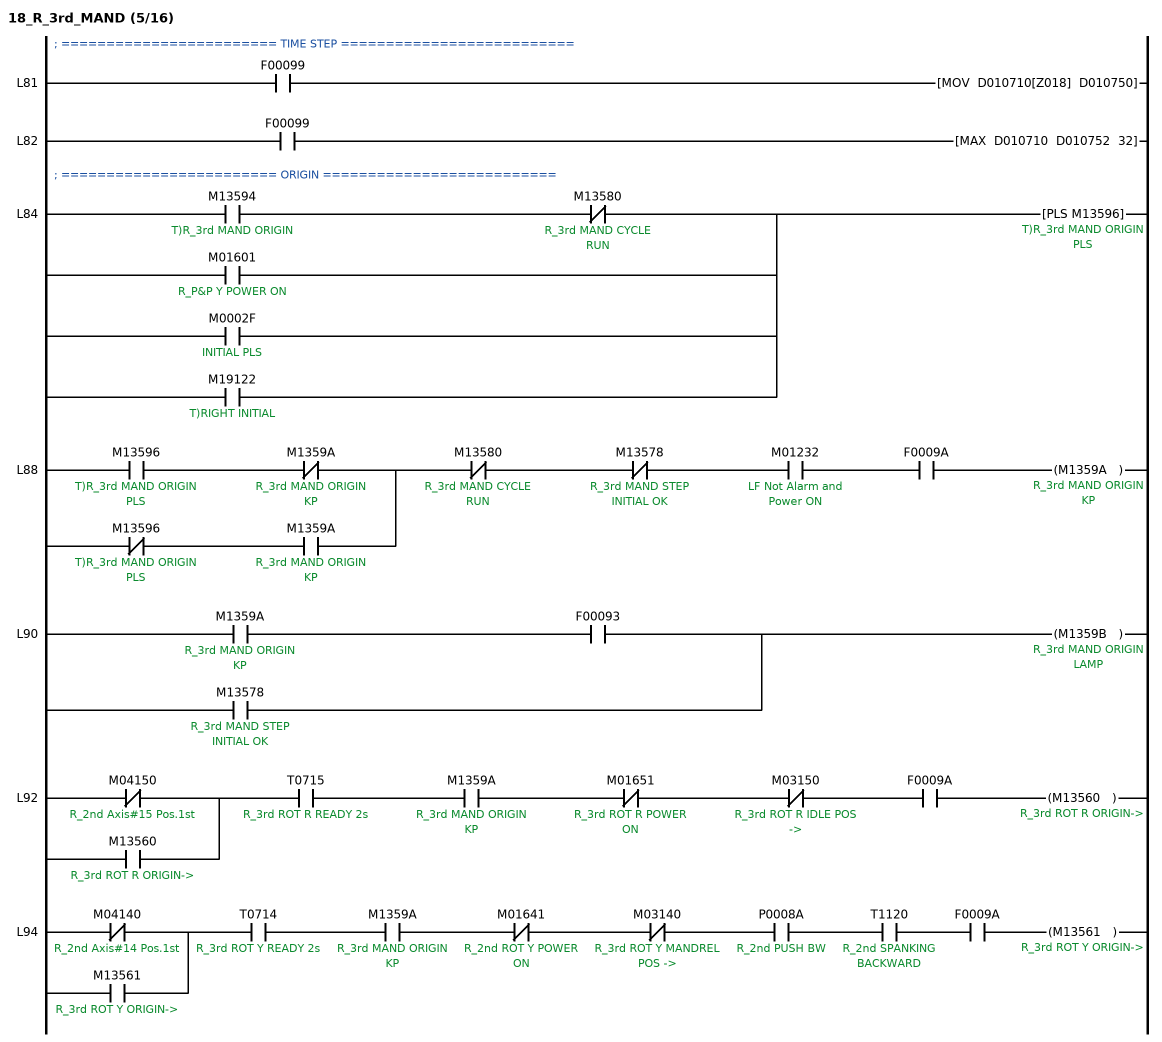
// ======================== TIME STEP ==========================
; L81
LOAD      F00099
MOV       D010710[Z018] D010750
; L82
LOAD      F00099
MAX       D010710 D010752 32
// ======================== ORIGIN ==========================
; L84
LOAD      M13594	// T)R_3rd MAND ORIGIN
AND NOT   M13580	// R_3rd MAND CYCLE RUN
OR        M01601	// R_P&P Y POWER ON
OR        M0002F	// INITIAL PLS
OR        M19122	// T)RIGHT INITIAL
OUTP      M13596	// T)R_3rd MAND ORIGIN PLS
; L88
LOAD      M13596	// T)R_3rd MAND ORIGIN PLS
AND NOT   M1359A	// R_3rd MAND ORIGIN KP
LOAD NOT  M13596	// T)R_3rd MAND ORIGIN PLS
AND       M1359A	// R_3rd MAND ORIGIN KP
OR LOAD
AND NOT   M13580	// R_3rd MAND CYCLE RUN
AND NOT   M13578	// R_3rd MAND STEP INITIAL OK
AND       M01232	// LF Not Alarm and Power ON
AND       F0009A
OUT       M1359A	// R_3rd MAND ORIGIN KP
; L90
LOAD      M1359A	// R_3rd MAND ORIGIN KP
AND       F00093
OR        M13578	// R_3rd MAND STEP INITIAL OK
OUT       M1359B	// R_3rd MAND ORIGIN LAMP
; L92
LOAD NOT  M04150	// R_2nd Axis#15 Pos.1st
OR        M13560	// R_3rd ROT R ORIGIN->
AND       T0715	// R_3rd ROT R READY 2s
AND       M1359A	// R_3rd MAND ORIGIN KP
AND NOT   M01651	// R_3rd ROT R POWER ON
AND NOT   M03150	// R_3rd ROT R IDLE POS ->
AND       F0009A
OUT       M13560	// R_3rd ROT R ORIGIN->
; L94
LOAD NOT  M04140	// R_2nd Axis#14 Pos.1st
OR        M13561	// R_3rd ROT Y ORIGIN->
AND       T0714	// R_3rd ROT Y READY 2s
AND       M1359A	// R_3rd MAND ORIGIN KP
AND NOT   M01641	// R_2nd ROT Y POWER ON
AND NOT   M03140	// R_3rd ROT Y MANDREL POS ->
AND       P0008A	// R_2nd PUSH BW
AND       T1120	// R_2nd SPANKING BACKWARD
AND       F0009A
OUT       M13561	// R_3rd ROT Y ORIGIN->

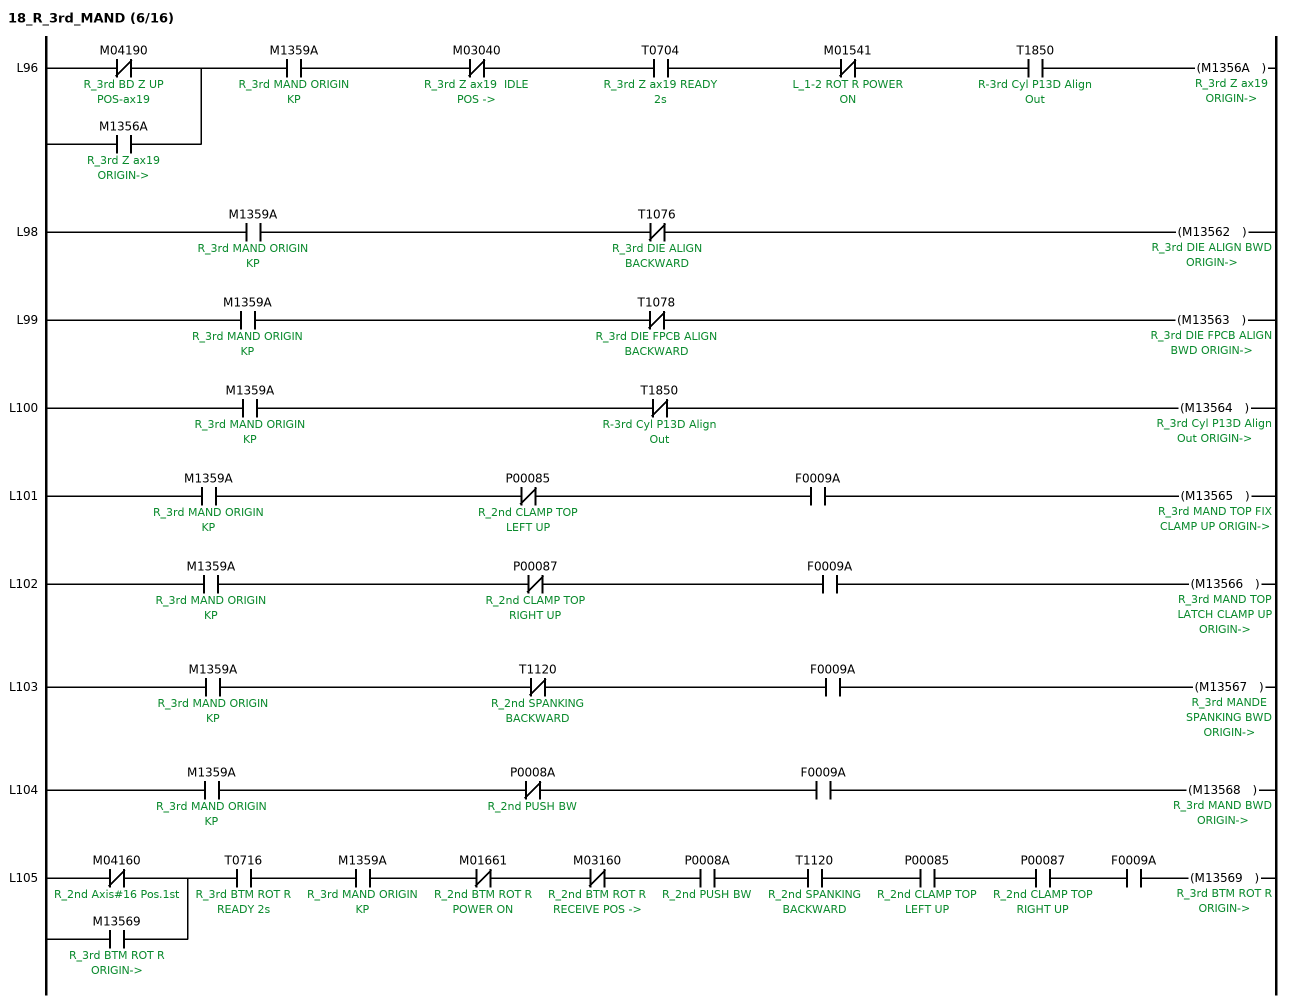
; L96
LOAD NOT  M04190	// R_3rd BD Z UP POS-ax19
OR        M1356A	// R_3rd Z ax19 ORIGIN->
AND       M1359A	// R_3rd MAND ORIGIN KP
AND NOT   M03040	// R_3rd Z ax19  IDLE POS ->
AND       T0704	// R_3rd Z ax19 READY 2s
AND NOT   M01541	// L_1-2 ROT R POWER ON
AND       T1850	// R-3rd Cyl P13D Align Out
OUT       M1356A	// R_3rd Z ax19 ORIGIN->
; L98
LOAD      M1359A	// R_3rd MAND ORIGIN KP
AND NOT   T1076	// R_3rd DIE ALIGN BACKWARD
OUT       M13562	// R_3rd DIE ALIGN BWD ORIGIN->
; L99
LOAD      M1359A	// R_3rd MAND ORIGIN KP
AND NOT   T1078	// R_3rd DIE FPCB ALIGN BACKWARD
OUT       M13563	// R_3rd DIE FPCB ALIGN BWD ORIGIN->
; L100
LOAD      M1359A	// R_3rd MAND ORIGIN KP
AND NOT   T1850	// R-3rd Cyl P13D Align Out
OUT       M13564	// R_3rd Cyl P13D Align Out ORIGIN->
; L101
LOAD      M1359A	// R_3rd MAND ORIGIN KP
AND NOT   P00085	// R_2nd CLAMP TOP LEFT UP
AND       F0009A
OUT       M13565	// R_3rd MAND TOP FIX CLAMP UP ORIGIN->
; L102
LOAD      M1359A	// R_3rd MAND ORIGIN KP
AND NOT   P00087	// R_2nd CLAMP TOP RIGHT UP
AND       F0009A
OUT       M13566	// R_3rd MAND TOP LATCH CLAMP UP ORIGIN->
; L103
LOAD      M1359A	// R_3rd MAND ORIGIN KP
AND NOT   T1120	// R_2nd SPANKING BACKWARD
AND       F0009A
OUT       M13567	// R_3rd MANDE SPANKING BWD ORIGIN->
; L104
LOAD      M1359A	// R_3rd MAND ORIGIN KP
AND NOT   P0008A	// R_2nd PUSH BW
AND       F0009A
OUT       M13568	// R_3rd MAND BWD ORIGIN->
; L105
LOAD NOT  M04160	// R_2nd Axis#16 Pos.1st
OR        M13569	// R_3rd BTM ROT R ORIGIN->
AND       T0716	// R_3rd BTM ROT R READY 2s
AND       M1359A	// R_3rd MAND ORIGIN KP
AND NOT   M01661	// R_2nd BTM ROT R POWER ON
AND NOT   M03160	// R_2nd BTM ROT R RECEIVE POS ->
AND       P0008A	// R_2nd PUSH BW
AND       T1120	// R_2nd SPANKING BACKWARD
AND       P00085	// R_2nd CLAMP TOP LEFT UP
AND       P00087	// R_2nd CLAMP TOP RIGHT UP
AND       F0009A
OUT       M13569	// R_3rd BTM ROT R ORIGIN->

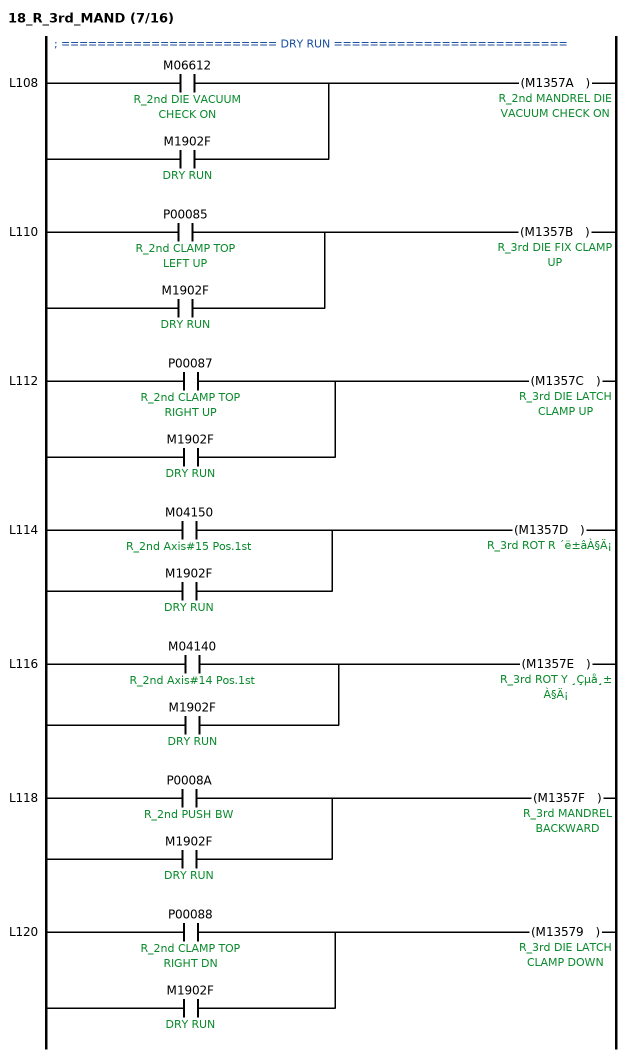
// ======================== DRY RUN ==========================
; L108
LOAD      M06612	// R_2nd DIE VACUUM CHECK ON
OR        M1902F	// DRY RUN
OUT       M1357A	// R_2nd MANDREL DIE VACUUM CHECK ON
; L110
LOAD      P00085	// R_2nd CLAMP TOP LEFT UP
OR        M1902F	// DRY RUN
OUT       M1357B	// R_3rd DIE FIX CLAMP UP
; L112
LOAD      P00087	// R_2nd CLAMP TOP RIGHT UP
OR        M1902F	// DRY RUN
OUT       M1357C	// R_3rd DIE LATCH CLAMP UP
; L114
LOAD      M04150	// R_2nd Axis#15 Pos.1st
OR        M1902F	// DRY RUN
OUT       M1357D	// R_3rd ROT R ´ë±âÀ§Ä¡
; L116
LOAD      M04140	// R_2nd Axis#14 Pos.1st
OR        M1902F	// DRY RUN
OUT       M1357E	// R_3rd ROT Y ¸Çµå¸± À§Ä¡
; L118
LOAD      P0008A	// R_2nd PUSH BW
OR        M1902F	// DRY RUN
OUT       M1357F	// R_3rd MANDREL BACKWARD
; L120
LOAD      P00088	// R_2nd CLAMP TOP RIGHT DN
OR        M1902F	// DRY RUN
OUT       M13579	// R_3rd DIE LATCH CLAMP DOWN

